(* CODESYS project mobject-graph-vision-pack.library
   Company: mobject
   Version: 0.5.0
   DefaultNamespace: mobject-graph-vision-pack
   Title: mobject-graph-vision-pack
   Placeholder: mobject-graph-vision-pack
   Author: mobject dev team
   DocFormat: reStructuredText

Project tree, tasks and I/O mapping:
  libraries: mobject-core, 0.3.0 (mobject); mobject-graph, 0.11.0 (mobject); mobject-graph-plc-pack, 0.12.0 (mobject); Tc2_Standard, * (Beckhoff Automation GmbH); Tc2_System, * (Beckhoff Automation GmbH); Tc3_Module, * (Beckhoff Automation GmbH); Tc3_Vision, * (Beckhoff Automation GmbH)
  Datatypes/
    Aliases/
    Arrays/
    Enums/
      function block _ETcVn2dCodeSearchStrategy [ST]: FB_init, AddLocalEnumeration, IsEnumeratorValueEqual, SetBaseDatatypeReference, Address, ClearReference, Clone, Identifier, MakeReferenceTo, Size, TryMakeReferenceTo, Value
      function block _ETcVnAdaptiveThresholdMethod [ST]: FB_init, AddLocalEnumeration, IsEnumeratorValueEqual, SetBaseDatatypeReference, Address, ClearReference, Clone, Identifier, MakeReferenceTo, Size, TryMakeReferenceTo, Value
      function block _ETcVnBarcodeSearchDirection [ST]: FB_init, AddLocalEnumeration, IsEnumeratorValueEqual, SetBaseDatatypeReference, Address, ClearReference, Clone, Identifier, MakeReferenceTo, Size, TryMakeReferenceTo, Value
      function block _ETcVnBarcodeType [ST]: FB_init, AddLocalEnumeration, IsEnumeratorValueEqual, SetBaseDatatypeReference, Address, ClearReference, Clone, Identifier, MakeReferenceTo, Size, TryMakeReferenceTo, Value
      function block _ETcVnBlobCombination [ST]: FB_init, AddLocalEnumeration, IsEnumeratorValueEqual, SetBaseDatatypeReference, Address, ClearReference, Clone, Identifier, MakeReferenceTo, Size, TryMakeReferenceTo, Value
      function block _ETcVnBorderInterpolationMethod [ST]: FB_init, AddLocalEnumeration, IsEnumeratorValueEqual, SetBaseDatatypeReference, Address, ClearReference, Clone, Identifier, MakeReferenceTo, Size, TryMakeReferenceTo, Value
      function block _ETcVnCalibrationPattern [ST]: FB_init, AddLocalEnumeration, IsEnumeratorValueEqual, SetBaseDatatypeReference, Address, ClearReference, Clone, Identifier, MakeReferenceTo, Size, TryMakeReferenceTo, Value
      function block _ETcVnCalibrationPatternOrigin [ST]: FB_init, AddLocalEnumeration, IsEnumeratorValueEqual, SetBaseDatatypeReference, Address, ClearReference, Clone, Identifier, MakeReferenceTo, Size, TryMakeReferenceTo, Value
      function block _ETcVnCameraState [ST]: FB_init, AddLocalEnumeration, IsEnumeratorValueEqual, SetBaseDatatypeReference, Address, ClearReference, Clone, Identifier, MakeReferenceTo, Size, TryMakeReferenceTo, Value
      function block _ETcVnClusteringAlgorithm [ST]: FB_init, AddLocalEnumeration, IsEnumeratorValueEqual, SetBaseDatatypeReference, Address, ClearReference, Clone, Identifier, MakeReferenceTo, Size, TryMakeReferenceTo, Value
      function block _ETcVnColorMap [ST]: FB_init, AddLocalEnumeration, IsEnumeratorValueEqual, SetBaseDatatypeReference, Address, ClearReference, Clone, Identifier, MakeReferenceTo, Size, TryMakeReferenceTo, Value
      function block _ETcVnColorMapSize [ST]: FB_init, AddLocalEnumeration, IsEnumeratorValueEqual, SetBaseDatatypeReference, Address, ClearReference, Clone, Identifier, MakeReferenceTo, Size, TryMakeReferenceTo, Value
      function block _ETcVnColorSpaceTransform [ST]: FB_init, AddLocalEnumeration, IsEnumeratorValueEqual, SetBaseDatatypeReference, Address, ClearReference, Clone, Identifier, MakeReferenceTo, Size, TryMakeReferenceTo, Value
      function block _ETcVnColorTrainingMethod [ST]: FB_init, AddLocalEnumeration, IsEnumeratorValueEqual, SetBaseDatatypeReference, Address, ClearReference, Clone, Identifier, MakeReferenceTo, Size, TryMakeReferenceTo, Value
      function block _ETcVnConnectedComponentsAlgorithm [ST]: FB_init, AddLocalEnumeration, IsEnumeratorValueEqual, SetBaseDatatypeReference, Address, ClearReference, Clone, Identifier, MakeReferenceTo, Size, TryMakeReferenceTo, Value
      function block _ETcVnContainerExportFormat [ST]: FB_init, AddLocalEnumeration, IsEnumeratorValueEqual, SetBaseDatatypeReference, Address, ClearReference, Clone, Identifier, MakeReferenceTo, Size, TryMakeReferenceTo, Value
      function block _ETcVnContourApproximationMethod [ST]: FB_init, AddLocalEnumeration, IsEnumeratorValueEqual, SetBaseDatatypeReference, Address, ClearReference, Clone, Identifier, MakeReferenceTo, Size, TryMakeReferenceTo, Value
      function block _ETcVnContourRetrievalMode [ST]: FB_init, AddLocalEnumeration, IsEnumeratorValueEqual, SetBaseDatatypeReference, Address, ClearReference, Clone, Identifier, MakeReferenceTo, Size, TryMakeReferenceTo, Value
      function block _ETcVnContoursMatchComparisonMethod [ST]: FB_init, AddLocalEnumeration, IsEnumeratorValueEqual, SetBaseDatatypeReference, Address, ClearReference, Clone, Identifier, MakeReferenceTo, Size, TryMakeReferenceTo, Value
      function block _ETcVnDiffusivityTypeKAZE [ST]: FB_init, AddLocalEnumeration, IsEnumeratorValueEqual, SetBaseDatatypeReference, Address, ClearReference, Clone, Identifier, MakeReferenceTo, Size, TryMakeReferenceTo, Value
      function block _ETcVnDistanceTransformationLabel [ST]: FB_init, AddLocalEnumeration, IsEnumeratorValueEqual, SetBaseDatatypeReference, Address, ClearReference, Clone, Identifier, MakeReferenceTo, Size, TryMakeReferenceTo, Value
      function block _ETcVnDistanceTransformationMask [ST]: FB_init, AddLocalEnumeration, IsEnumeratorValueEqual, SetBaseDatatypeReference, Address, ClearReference, Clone, Identifier, MakeReferenceTo, Size, TryMakeReferenceTo, Value
      function block _ETcVnDistanceType [ST]: FB_init, AddLocalEnumeration, IsEnumeratorValueEqual, SetBaseDatatypeReference, Address, ClearReference, Clone, Identifier, MakeReferenceTo, Size, TryMakeReferenceTo, Value
      function block _ETcVnDrawMatchesFlags [ST]: FB_init, AddLocalEnumeration, IsEnumeratorValueEqual, SetBaseDatatypeReference, Address, ClearReference, Clone, Identifier, MakeReferenceTo, Size, TryMakeReferenceTo, Value
      function block _ETcVnDrawShape [ST]: FB_init, AddLocalEnumeration, IsEnumeratorValueEqual, SetBaseDatatypeReference, Address, ClearReference, Clone, Identifier, MakeReferenceTo, Size, TryMakeReferenceTo, Value
      function block _ETcVnEdgeDetectionAlgorithm [ST]: FB_init, AddLocalEnumeration, IsEnumeratorValueEqual, SetBaseDatatypeReference, Address, ClearReference, Clone, Identifier, MakeReferenceTo, Size, TryMakeReferenceTo, Value
      function block _ETcVnEdgeDirection [ST]: FB_init, AddLocalEnumeration, IsEnumeratorValueEqual, SetBaseDatatypeReference, Address, ClearReference, Clone, Identifier, MakeReferenceTo, Size, TryMakeReferenceTo, Value
      function block _ETcVnElementType [ST]: FB_init, AddLocalEnumeration, IsEnumeratorValueEqual, SetBaseDatatypeReference, Address, ClearReference, Clone, Identifier, MakeReferenceTo, Size, TryMakeReferenceTo, Value
      function block _ETcVnEstimationAlgorithm [ST]: FB_init, AddLocalEnumeration, IsEnumeratorValueEqual, SetBaseDatatypeReference, Address, ClearReference, Clone, Identifier, MakeReferenceTo, Size, TryMakeReferenceTo, Value
      function block _ETcVnExtremePointDirection [ST]: FB_init, AddLocalEnumeration, IsEnumeratorValueEqual, SetBaseDatatypeReference, Address, ClearReference, Clone, Identifier, MakeReferenceTo, Size, TryMakeReferenceTo, Value
      function block _ETcVnFeatureDescriptorTypeAKAZE [ST]: FB_init, AddLocalEnumeration, IsEnumeratorValueEqual, SetBaseDatatypeReference, Address, ClearReference, Clone, Identifier, MakeReferenceTo, Size, TryMakeReferenceTo, Value
      function block _ETcVnFeatureScoreTypeORB [ST]: FB_init, AddLocalEnumeration, IsEnumeratorValueEqual, SetBaseDatatypeReference, Address, ClearReference, Clone, Identifier, MakeReferenceTo, Size, TryMakeReferenceTo, Value
      function block _ETcVnFilterDirection [ST]: FB_init, AddLocalEnumeration, IsEnumeratorValueEqual, SetBaseDatatypeReference, Address, ClearReference, Clone, Identifier, MakeReferenceTo, Size, TryMakeReferenceTo, Value
      function block _ETcVnFlipAxis [ST]: FB_init, AddLocalEnumeration, IsEnumeratorValueEqual, SetBaseDatatypeReference, Address, ClearReference, Clone, Identifier, MakeReferenceTo, Size, TryMakeReferenceTo, Value
      function block _ETcVnFontType [ST]: FB_init, AddLocalEnumeration, IsEnumeratorValueEqual, SetBaseDatatypeReference, Address, ClearReference, Clone, Identifier, MakeReferenceTo, Size, TryMakeReferenceTo, Value
      function block _ETcVnHoughMethod [ST]: FB_init, AddLocalEnumeration, IsEnumeratorValueEqual, SetBaseDatatypeReference, Address, ClearReference, Clone, Identifier, MakeReferenceTo, Size, TryMakeReferenceTo, Value
      function block _ETcVnInterpolationType [ST]: FB_init, AddLocalEnumeration, IsEnumeratorValueEqual, SetBaseDatatypeReference, Address, ClearReference, Clone, Identifier, MakeReferenceTo, Size, TryMakeReferenceTo, Value
      function block _ETcVnKeypointDetectionTypeAGAST [ST]: FB_init, AddLocalEnumeration, IsEnumeratorValueEqual, SetBaseDatatypeReference, Address, ClearReference, Clone, Identifier, MakeReferenceTo, Size, TryMakeReferenceTo, Value
      function block _ETcVnKeypointDetectionTypeFAST [ST]: FB_init, AddLocalEnumeration, IsEnumeratorValueEqual, SetBaseDatatypeReference, Address, ClearReference, Clone, Identifier, MakeReferenceTo, Size, TryMakeReferenceTo, Value
      function block _ETcVnLineType [ST]: FB_init, AddLocalEnumeration, IsEnumeratorValueEqual, SetBaseDatatypeReference, Address, ClearReference, Clone, Identifier, MakeReferenceTo, Size, TryMakeReferenceTo, Value
      function block _ETcVnMorphologicalOperator [ST]: FB_init, AddLocalEnumeration, IsEnumeratorValueEqual, SetBaseDatatypeReference, Address, ClearReference, Clone, Identifier, MakeReferenceTo, Size, TryMakeReferenceTo, Value
      function block _ETcVnNormalizationType [ST]: FB_init, AddLocalEnumeration, IsEnumeratorValueEqual, SetBaseDatatypeReference, Address, ClearReference, Clone, Identifier, MakeReferenceTo, Size, TryMakeReferenceTo, Value
      function block _ETcVnOrientationMethod [ST]: FB_init, AddLocalEnumeration, IsEnumeratorValueEqual, SetBaseDatatypeReference, Address, ClearReference, Clone, Identifier, MakeReferenceTo, Size, TryMakeReferenceTo, Value
      function block _ETcVnPixelConnectivity [ST]: FB_init, AddLocalEnumeration, IsEnumeratorValueEqual, SetBaseDatatypeReference, Address, ClearReference, Clone, Identifier, MakeReferenceTo, Size, TryMakeReferenceTo, Value
      function block _ETcVnPixelEncoding [ST]: FB_init, AddLocalEnumeration, IsEnumeratorValueEqual, SetBaseDatatypeReference, Address, ClearReference, Clone, Identifier, MakeReferenceTo, Size, TryMakeReferenceTo, Value
      function block _ETcVnPixelPackMode [ST]: FB_init, AddLocalEnumeration, IsEnumeratorValueEqual, SetBaseDatatypeReference, Address, ClearReference, Clone, Identifier, MakeReferenceTo, Size, TryMakeReferenceTo, Value
      function block _ETcVnRectangleIntersection [ST]: FB_init, AddLocalEnumeration, IsEnumeratorValueEqual, SetBaseDatatypeReference, Address, ClearReference, Clone, Identifier, MakeReferenceTo, Size, TryMakeReferenceTo, Value
      function block _ETcVnRotationAngle [ST]: FB_init, AddLocalEnumeration, IsEnumeratorValueEqual, SetBaseDatatypeReference, Address, ClearReference, Clone, Identifier, MakeReferenceTo, Size, TryMakeReferenceTo, Value
      function block _ETcVnSignedNormalization [ST]: FB_init, AddLocalEnumeration, IsEnumeratorValueEqual, SetBaseDatatypeReference, Address, ClearReference, Clone, Identifier, MakeReferenceTo, Size, TryMakeReferenceTo, Value
      function block _ETcVnStructuringElementShape [ST]: FB_init, AddLocalEnumeration, IsEnumeratorValueEqual, SetBaseDatatypeReference, Address, ClearReference, Clone, Identifier, MakeReferenceTo, Size, TryMakeReferenceTo, Value
      function block _ETcVnTemplateMatchMethod [ST]: FB_init, AddLocalEnumeration, IsEnumeratorValueEqual, SetBaseDatatypeReference, Address, ClearReference, Clone, Identifier, MakeReferenceTo, Size, TryMakeReferenceTo, Value
      function block _ETcVnThresholdType [ST]: FB_init, AddLocalEnumeration, IsEnumeratorValueEqual, SetBaseDatatypeReference, Address, ClearReference, Clone, Identifier, MakeReferenceTo, Size, TryMakeReferenceTo, Value
      function block _ETcVnVectorCompareMethod [ST]: FB_init, AddLocalEnumeration, IsEnumeratorValueEqual, SetBaseDatatypeReference, Address, ClearReference, Clone, Identifier, MakeReferenceTo, Size, TryMakeReferenceTo, Value
      function block _ETcVnWorldCoordinateSystem [ST]: FB_init, AddLocalEnumeration, IsEnumeratorValueEqual, SetBaseDatatypeReference, Address, ClearReference, Clone, Identifier, MakeReferenceTo, Size, TryMakeReferenceTo, Value
      function block _ETcWatchdogAccumulationType [ST]: FB_init, AddLocalEnumeration, IsEnumeratorValueEqual, SetBaseDatatypeReference, Address, ClearReference, Clone, Identifier, MakeReferenceTo, Size, TryMakeReferenceTo, Value
      function block _GEV_CAMERA_STATE [ST]: FB_init, AddLocalEnumeration, IsEnumeratorValueEqual, SetBaseDatatypeReference, Address, ClearReference, Clone, Identifier, MakeReferenceTo, Size, TryMakeReferenceTo, Value
    Interface/
      function block _ITcVnImage [ST]: TryGetElementTypeFromInfo, Address, ClearReference, Clone, Identifier, MakeReferenceTo, SerializeWith, Size, TryDeserializeFrom, TryMakeReferenceTo, Value
    Structs/
      function block _TcVnImageInfo [ST]: FB_init, SetMemberReference, Address, ClearReference, Clone, Identifier, MakeReferenceTo, nHeight, nImageSize, nWidth, nXPadding, nYPadding, Size, stPixelFormat, TryMakeReferenceTo, Value
      function block _TcVnPixelFormat [ST]: FB_init, SetMemberReference, Address, bFloat, bPlanar, bSigned, bSupported, ClearReference, Clone, ePixelEncoding, ePixelPackMode, Identifier, MakeReferenceTo, nChannels, nElementSize, nTotalSize, Size, TryMakeReferenceTo, Value
    function block VisionDatatypePack [ST]: RegisterWithDatatypes
  Nodes/
    Image Filtering/
      function block Node_F_VN_GaussianFilter [ST]: FB_init, Clone, OnExecute
    function block VisionNodePack [ST]: RegisterWithNodeFactory
  function block VisionPack [ST]: RegisterWithDatatypes, RegisterWithNodeFactory
*)

// Datatypes/Enums/_ETcVn2dCodeSearchStrategy
{attribute 'linkalways'} 
{attribute 'no_explicit_call' := 'This FB is a CLASS and must be accessed using methods or properties'}
{attribute 'enable_dynamic_creation'}
FUNCTION_BLOCK _ETcVn2dCodeSearchStrategy EXTENDS EnumDatatypeBase
VAR
	localData : ETcVn2dCodeSearchStrategy;
	activeData : REFERENCE TO ETcVn2dCodeSearchStrategy;
	enumBaseDatatype : _UDINT(localData);
END_VAR

METHOD FB_init : BOOL
VAR_INPUT
	bInitRetains : BOOL; // if TRUE, the retain variables are initialized (warm start / cold start)
	bInCopyCode : BOOL;  // if TRUE, the instance afterwards gets moved into the copy code (online change)
	InitialValue : ETcVn2dCodeSearchStrategy;
END_VAR
localData := InitialValue;
AddBaseDatatype(enumBaseDatatype);
ClearReference();

AddLocalEnumeration('TCVN_CSS_DEFAULT', ETcVn2dCodeSearchStrategy.TCVN_CSS_DEFAULT);
AddLocalEnumeration('TCVN_CSS_FIRST_FLIPPED', ETcVn2dCodeSearchStrategy.TCVN_CSS_FIRST_FLIPPED);
AddLocalEnumeration('TCVN_CSS_FIRST_INVERTED', ETcVn2dCodeSearchStrategy.TCVN_CSS_FIRST_INVERTED);
AddLocalEnumeration('TCVN_CSS_FIRST_NOT_FLIPPED', ETcVn2dCodeSearchStrategy.TCVN_CSS_FIRST_NOT_FLIPPED);
AddLocalEnumeration('TCVN_CSS_FIRST_NOT_INVERTED', ETcVn2dCodeSearchStrategy.TCVN_CSS_FIRST_NOT_INVERTED);
AddLocalEnumeration('TCVN_CSS_ONLY_FLIPPED', ETcVn2dCodeSearchStrategy.TCVN_CSS_ONLY_FLIPPED);
AddLocalEnumeration('TCVN_CSS_ONLY_INVERTED', ETcVn2dCodeSearchStrategy.TCVN_CSS_ONLY_INVERTED);
AddLocalEnumeration('TCVN_CSS_ONLY_NOT_FLIPPED', ETcVn2dCodeSearchStrategy.TCVN_CSS_ONLY_NOT_FLIPPED);
AddLocalEnumeration('TCVN_CSS_ONLY_NOT_INVERTED', ETcVn2dCodeSearchStrategy.TCVN_CSS_ONLY_NOT_INVERTED);
END_METHOD

METHOD PRIVATE AddLocalEnumeration
VAR_INPUT
	Enumeration : T_MAXSTRING;
	Value : ETcVn2dCodeSearchStrategy;
END_VAR
AddEnumeration(Enumeration, Value);
END_METHOD

METHOD IsEnumeratorValueEqual : BOOL
VAR_INPUT
	Enumerator : I_KeyValueForwardEnumerator;
END_VAR
VAR
	storedValue : ETcVn2dCodeSearchStrategy;
END_VAR
IF NOT Enumerator.TryGet(storedValue) THEN
	RETURN;
END_IF

IsEnumeratorValueEqual := storedValue = activeData;
END_METHOD

METHOD PROTECTED SetBaseDatatypeReference
VAR_INPUT
END_VAR
enumBaseDatatype.MakeReferenceTo(activeData);
END_METHOD

PROPERTY PUBLIC Address : PVOID
GET
Address := ADR(activeData);
END_GET
END_PROPERTY

METHOD PUBLIC ClearReference
VAR_INPUT
END_VAR
activeData REF= localData;
SetBaseDatatypeReference();
END_METHOD

METHOD PUBLIC Clone : I_Datatype
VAR
    pClone : POINTER TO _ETcVn2dCodeSearchStrategy;
END_VAR
pClone := __NEW(_ETcVn2dCodeSearchStrategy(InitialValue := Value));
Clone := pClone^;
END_METHOD

PROPERTY PUBLIC Identifier : T_MAXSTRING
GET
Identifier := 'ETcVn2dCodeSearchStrategy';
END_GET
END_PROPERTY

METHOD PUBLIC MakeReferenceTo
VAR_INPUT
	ReferenceTarget : REFERENCE TO ETcVn2dCodeSearchStrategy;
END_VAR
activeData REF= ReferenceTarget;
SetBaseDatatypeReference();
END_METHOD

PROPERTY PUBLIC Size : UDINT
GET
Size := SIZEOF(activeData);
END_GET
END_PROPERTY

METHOD TryMakeReferenceTo : BOOL
VAR_INPUT
	Target : I_Datatype;
END_VAR
VAR
	targetAsEnum : I_EnumDatatype;
	pTargetData : POINTER TO ETcVn2dCodeSearchStrategy;
END_VAR
IF NOT Target.TryResolveAsEnumDatatype(targetAsEnum) THEN
	RETURN;
END_IF

IF targetAsEnum.Identifier <> Identifier THEN
	RETURN;
END_IF

pTargetData := Target.Address;
activeData REF= pTargetData^;
SetBaseDatatypeReference();
TryMakeReferenceTo := TRUE;
END_METHOD

PROPERTY PUBLIC Value : ETcVn2dCodeSearchStrategy
GET
Value := activeData;
END_GET
SET
activeData := Value;
END_SET
END_PROPERTY

END_FUNCTION_BLOCK

// Datatypes/Enums/_ETcVnAdaptiveThresholdMethod
{attribute 'linkalways'} 
{attribute 'no_explicit_call' := 'This FB is a CLASS and must be accessed using methods or properties'}
{attribute 'enable_dynamic_creation'}
FUNCTION_BLOCK _ETcVnAdaptiveThresholdMethod EXTENDS EnumDatatypeBase
VAR
	localData : ETcVnAdaptiveThresholdMethod;
	activeData : REFERENCE TO ETcVnAdaptiveThresholdMethod;
	enumBaseDatatype : _DINT(localData);
END_VAR

METHOD FB_init : BOOL
VAR_INPUT
	bInitRetains : BOOL; // if TRUE, the retain variables are initialized (warm start / cold start)
	bInCopyCode : BOOL;  // if TRUE, the instance afterwards gets moved into the copy code (online change)
	InitialValue : ETcVnAdaptiveThresholdMethod;
END_VAR
localData := InitialValue;
AddBaseDatatype(enumBaseDatatype);
ClearReference();

AddLocalEnumeration('TCVN_ATM_MEAN', ETcVnAdaptiveThresholdMethod.TCVN_ATM_MEAN);
AddLocalEnumeration('TCVN_ATM_GAUSSIAN', ETcVnAdaptiveThresholdMethod.TCVN_ATM_GAUSSIAN);
END_METHOD

METHOD PRIVATE AddLocalEnumeration
VAR_INPUT
	Enumeration : T_MAXSTRING;
	Value : ETcVnAdaptiveThresholdMethod;
END_VAR
AddEnumeration(Enumeration, Value);
END_METHOD

METHOD IsEnumeratorValueEqual : BOOL
VAR_INPUT
	Enumerator : I_KeyValueForwardEnumerator;
END_VAR
VAR
	storedValue : ETcVnAdaptiveThresholdMethod;
END_VAR
IF NOT Enumerator.TryGet(storedValue) THEN
	RETURN;
END_IF

IsEnumeratorValueEqual := storedValue = activeData;
END_METHOD

METHOD PROTECTED SetBaseDatatypeReference
VAR_INPUT
END_VAR
enumBaseDatatype.MakeReferenceTo(activeData);
END_METHOD

PROPERTY PUBLIC Address : PVOID
GET
Address := ADR(activeData);
END_GET
END_PROPERTY

METHOD PUBLIC ClearReference
VAR_INPUT
END_VAR
activeData REF= localData;
SetBaseDatatypeReference();
END_METHOD

METHOD PUBLIC Clone : I_Datatype
VAR
    pClone : POINTER TO _ETcVnAdaptiveThresholdMethod;
END_VAR
pClone := __NEW(_ETcVnAdaptiveThresholdMethod(InitialValue := Value));
Clone := pClone^;
END_METHOD

PROPERTY PUBLIC Identifier : T_MAXSTRING
GET
Identifier := 'ETcVnAdaptiveThresholdMethod';
END_GET
END_PROPERTY

METHOD PUBLIC MakeReferenceTo
VAR_INPUT
	ReferenceTarget : REFERENCE TO ETcVnAdaptiveThresholdMethod;
END_VAR
activeData REF= ReferenceTarget;
SetBaseDatatypeReference();
END_METHOD

PROPERTY PUBLIC Size : UDINT
GET
Size := SIZEOF(activeData);
END_GET
END_PROPERTY

METHOD TryMakeReferenceTo : BOOL
VAR_INPUT
	Target : I_Datatype;
END_VAR
VAR
	targetAsEnum : I_EnumDatatype;
	pTargetData : POINTER TO ETcVnAdaptiveThresholdMethod;
END_VAR
IF NOT Target.TryResolveAsEnumDatatype(targetAsEnum) THEN
	RETURN;
END_IF

IF targetAsEnum.Identifier <> Identifier THEN
	RETURN;
END_IF

pTargetData := Target.Address;
activeData REF= pTargetData^;
SetBaseDatatypeReference();
TryMakeReferenceTo := TRUE;
END_METHOD

PROPERTY PUBLIC Value : ETcVnAdaptiveThresholdMethod
GET
Value := activeData;
END_GET
SET
activeData := Value;
END_SET
END_PROPERTY

END_FUNCTION_BLOCK

// Datatypes/Enums/_ETcVnBarcodeSearchDirection
{attribute 'linkalways'} 
{attribute 'no_explicit_call' := 'This FB is a CLASS and must be accessed using methods or properties'}
{attribute 'enable_dynamic_creation'}
FUNCTION_BLOCK _ETcVnBarcodeSearchDirection EXTENDS EnumDatatypeBase
VAR
	localData : ETcVnBarcodeSearchDirection;
	activeData : REFERENCE TO ETcVnBarcodeSearchDirection;
	enumBaseDatatype : _UDINT(localData);
END_VAR

METHOD FB_init : BOOL
VAR_INPUT
	bInitRetains : BOOL; // if TRUE, the retain variables are initialized (warm start / cold start)
	bInCopyCode : BOOL;  // if TRUE, the instance afterwards gets moved into the copy code (online change)
	InitialValue : ETcVnBarcodeSearchDirection;
END_VAR
localData := InitialValue;
AddBaseDatatype(enumBaseDatatype);
ClearReference();

AddLocalEnumeration('TCVN_BSD_ANY', ETcVnBarcodeSearchDirection.TCVN_BSD_ANY);
AddLocalEnumeration('TCVN_BSD_HORIZONTAL', ETcVnBarcodeSearchDirection.TCVN_BSD_HORIZONTAL);
AddLocalEnumeration('TCVN_BSD_VERTICAL', ETcVnBarcodeSearchDirection.TCVN_BSD_VERTICAL);
END_METHOD

METHOD PRIVATE AddLocalEnumeration
VAR_INPUT
	Enumeration : T_MAXSTRING;
	Value : ETcVnBarcodeSearchDirection;
END_VAR
AddEnumeration(Enumeration, Value);
END_METHOD

METHOD IsEnumeratorValueEqual : BOOL
VAR_INPUT
	Enumerator : I_KeyValueForwardEnumerator;
END_VAR
VAR
	storedValue : ETcVnBarcodeSearchDirection;
END_VAR
IF NOT Enumerator.TryGet(storedValue) THEN
	RETURN;
END_IF

IsEnumeratorValueEqual := storedValue = activeData;
END_METHOD

METHOD PROTECTED SetBaseDatatypeReference
VAR_INPUT
END_VAR
enumBaseDatatype.MakeReferenceTo(activeData);
END_METHOD

PROPERTY PUBLIC Address : PVOID
GET
Address := ADR(activeData);
END_GET
END_PROPERTY

METHOD PUBLIC ClearReference
VAR_INPUT
END_VAR
activeData REF= localData;
SetBaseDatatypeReference();
END_METHOD

METHOD PUBLIC Clone : I_Datatype
VAR
    pClone : POINTER TO _ETcVnBarcodeSearchDirection;
END_VAR
pClone := __NEW(_ETcVnBarcodeSearchDirection(InitialValue := Value));
Clone := pClone^;
END_METHOD

PROPERTY PUBLIC Identifier : T_MAXSTRING
GET
Identifier := 'ETcVnBarcodeSearchDirection';
END_GET
END_PROPERTY

METHOD PUBLIC MakeReferenceTo
VAR_INPUT
	ReferenceTarget : REFERENCE TO ETcVnBarcodeSearchDirection;
END_VAR
activeData REF= ReferenceTarget;
SetBaseDatatypeReference();
END_METHOD

PROPERTY PUBLIC Size : UDINT
GET
Size := SIZEOF(activeData);
END_GET
END_PROPERTY

METHOD TryMakeReferenceTo : BOOL
VAR_INPUT
	Target : I_Datatype;
END_VAR
VAR
	targetAsEnum : I_EnumDatatype;
	pTargetData : POINTER TO ETcVnBarcodeSearchDirection;
END_VAR
IF NOT Target.TryResolveAsEnumDatatype(targetAsEnum) THEN
	RETURN;
END_IF

IF targetAsEnum.Identifier <> Identifier THEN
	RETURN;
END_IF

pTargetData := Target.Address;
activeData REF= pTargetData^;
SetBaseDatatypeReference();
TryMakeReferenceTo := TRUE;
END_METHOD

PROPERTY PUBLIC Value : ETcVnBarcodeSearchDirection
GET
Value := activeData;
END_GET
SET
activeData := Value;
END_SET
END_PROPERTY

END_FUNCTION_BLOCK

// Datatypes/Enums/_ETcVnBarcodeType
{attribute 'linkalways'} 
{attribute 'no_explicit_call' := 'This FB is a CLASS and must be accessed using methods or properties'}
{attribute 'enable_dynamic_creation'}
FUNCTION_BLOCK _ETcVnBarcodeType EXTENDS EnumDatatypeBase
VAR
	localData : ETcVnBarcodeType;
	activeData : REFERENCE TO ETcVnBarcodeType;
	enumBaseDatatype : _UDINT(localData);
END_VAR

METHOD FB_init : BOOL
VAR_INPUT
	bInitRetains : BOOL; // if TRUE, the retain variables are initialized (warm start / cold start)
	bInCopyCode : BOOL;  // if TRUE, the instance afterwards gets moved into the copy code (online change)
	InitialValue : ETcVnBarcodeType;
END_VAR
localData := InitialValue;
AddBaseDatatype(enumBaseDatatype);
ClearReference();

AddLocalEnumeration('TCVN_BT_CODABAR', ETcVnBarcodeType.TCVN_BT_CODABAR);
AddLocalEnumeration('TCVN_BT_CODE39', ETcVnBarcodeType.TCVN_BT_CODE39);
AddLocalEnumeration('TCVN_BT_CODE93', ETcVnBarcodeType.TCVN_BT_CODE93);
AddLocalEnumeration('TCVN_BT_CODE128', ETcVnBarcodeType.TCVN_BT_CODE128);
AddLocalEnumeration('TCVN_BT_EAN8', ETcVnBarcodeType.TCVN_BT_EAN8);
AddLocalEnumeration('TCVN_BT_EAN13', ETcVnBarcodeType.TCVN_BT_EAN13);
AddLocalEnumeration('TCVN_BT_ITF', ETcVnBarcodeType.TCVN_BT_ITF);
AddLocalEnumeration('TCVN_BT_UPCA', ETcVnBarcodeType.TCVN_BT_UPCA);
AddLocalEnumeration('TCVN_BT_UPCE', ETcVnBarcodeType.TCVN_BT_UPCE);
AddLocalEnumeration('TCVN_BT_ANY', ETcVnBarcodeType.TCVN_BT_ANY);
AddLocalEnumeration('TCVN_BT_CODE39EXTENDED', ETcVnBarcodeType.TCVN_BT_CODE39EXTENDED);
END_METHOD

METHOD PRIVATE AddLocalEnumeration
VAR_INPUT
	Enumeration : T_MAXSTRING;
	Value : ETcVnBarcodeType;
END_VAR
AddEnumeration(Enumeration, Value);
END_METHOD

METHOD IsEnumeratorValueEqual : BOOL
VAR_INPUT
	Enumerator : I_KeyValueForwardEnumerator;
END_VAR
VAR
	storedValue : ETcVnBarcodeType;
END_VAR
IF NOT Enumerator.TryGet(storedValue) THEN
	RETURN;
END_IF

IsEnumeratorValueEqual := storedValue = activeData;
END_METHOD

METHOD PROTECTED SetBaseDatatypeReference
VAR_INPUT
END_VAR
enumBaseDatatype.MakeReferenceTo(activeData);
END_METHOD

PROPERTY PUBLIC Address : PVOID
GET
Address := ADR(activeData);
END_GET
END_PROPERTY

METHOD PUBLIC ClearReference
VAR_INPUT
END_VAR
activeData REF= localData;
SetBaseDatatypeReference();
END_METHOD

METHOD PUBLIC Clone : I_Datatype
VAR
    pClone : POINTER TO _ETcVnBarcodeType;
END_VAR
pClone := __NEW(_ETcVnBarcodeType(InitialValue := Value));
Clone := pClone^;
END_METHOD

PROPERTY PUBLIC Identifier : T_MAXSTRING
GET
Identifier := 'ETcVnBarcodeType';
END_GET
END_PROPERTY

METHOD PUBLIC MakeReferenceTo
VAR_INPUT
	ReferenceTarget : REFERENCE TO ETcVnBarcodeType;
END_VAR
activeData REF= ReferenceTarget;
SetBaseDatatypeReference();
END_METHOD

PROPERTY PUBLIC Size : UDINT
GET
Size := SIZEOF(activeData);
END_GET
END_PROPERTY

METHOD TryMakeReferenceTo : BOOL
VAR_INPUT
	Target : I_Datatype;
END_VAR
VAR
	targetAsEnum : I_EnumDatatype;
	pTargetData : POINTER TO ETcVnBarcodeType;
END_VAR
IF NOT Target.TryResolveAsEnumDatatype(targetAsEnum) THEN
	RETURN;
END_IF

IF targetAsEnum.Identifier <> Identifier THEN
	RETURN;
END_IF

pTargetData := Target.Address;
activeData REF= pTargetData^;
SetBaseDatatypeReference();
TryMakeReferenceTo := TRUE;
END_METHOD

PROPERTY PUBLIC Value : ETcVnBarcodeType
GET
Value := activeData;
END_GET
SET
activeData := Value;
END_SET
END_PROPERTY

END_FUNCTION_BLOCK

// Datatypes/Enums/_ETcVnBlobCombination
{attribute 'linkalways'} 
{attribute 'no_explicit_call' := 'This FB is a CLASS and must be accessed using methods or properties'}
{attribute 'enable_dynamic_creation'}
FUNCTION_BLOCK _ETcVnBlobCombination EXTENDS EnumDatatypeBase
VAR
	localData : ETcVnBlobCombination;
	activeData : REFERENCE TO ETcVnBlobCombination;
	enumBaseDatatype : _DINT(localData);
END_VAR

METHOD FB_init : BOOL
VAR_INPUT
	bInitRetains : BOOL; // if TRUE, the retain variables are initialized (warm start / cold start)
	bInCopyCode : BOOL;  // if TRUE, the instance afterwards gets moved into the copy code (online change)
	InitialValue : ETcVnBlobCombination;
END_VAR
localData := InitialValue;
AddBaseDatatype(enumBaseDatatype);
ClearReference();

AddLocalEnumeration('TCVN_BC_SMALLEST', ETcVnBlobCombination.TCVN_BC_SMALLEST);
AddLocalEnumeration('TCVN_BC_LARGEST', ETcVnBlobCombination.TCVN_BC_LARGEST);
AddLocalEnumeration('TCVN_BC_MIN_THRESHOLD', ETcVnBlobCombination.TCVN_BC_MIN_THRESHOLD);
AddLocalEnumeration('TCVN_BC_MAX_THRESHOLD', ETcVnBlobCombination.TCVN_BC_MAX_THRESHOLD);
AddLocalEnumeration('TCVN_BC_MEDIAN_THRESHOLD', ETcVnBlobCombination.TCVN_BC_MEDIAN_THRESHOLD);
END_METHOD

METHOD PRIVATE AddLocalEnumeration
VAR_INPUT
	Enumeration : T_MAXSTRING;
	Value : ETcVnBlobCombination;
END_VAR
AddEnumeration(Enumeration, Value);
END_METHOD

METHOD IsEnumeratorValueEqual : BOOL
VAR_INPUT
	Enumerator : I_KeyValueForwardEnumerator;
END_VAR
VAR
	storedValue : ETcVnBlobCombination;
END_VAR
IF NOT Enumerator.TryGet(storedValue) THEN
	RETURN;
END_IF

IsEnumeratorValueEqual := storedValue = activeData;
END_METHOD

METHOD PROTECTED SetBaseDatatypeReference
VAR_INPUT
END_VAR
enumBaseDatatype.MakeReferenceTo(activeData);
END_METHOD

PROPERTY PUBLIC Address : PVOID
GET
Address := ADR(activeData);
END_GET
END_PROPERTY

METHOD PUBLIC ClearReference
VAR_INPUT
END_VAR
activeData REF= localData;
SetBaseDatatypeReference();
END_METHOD

METHOD PUBLIC Clone : I_Datatype
VAR
    pClone : POINTER TO _ETcVnBlobCombination;
END_VAR
pClone := __NEW(_ETcVnBlobCombination(InitialValue := Value));
Clone := pClone^;
END_METHOD

PROPERTY PUBLIC Identifier : T_MAXSTRING
GET
Identifier := 'ETcVnBlobCombination';
END_GET
END_PROPERTY

METHOD PUBLIC MakeReferenceTo
VAR_INPUT
	ReferenceTarget : REFERENCE TO ETcVnBlobCombination;
END_VAR
activeData REF= ReferenceTarget;
SetBaseDatatypeReference();
END_METHOD

PROPERTY PUBLIC Size : UDINT
GET
Size := SIZEOF(activeData);
END_GET
END_PROPERTY

METHOD TryMakeReferenceTo : BOOL
VAR_INPUT
	Target : I_Datatype;
END_VAR
VAR
	targetAsEnum : I_EnumDatatype;
	pTargetData : POINTER TO ETcVnBlobCombination;
END_VAR
IF NOT Target.TryResolveAsEnumDatatype(targetAsEnum) THEN
	RETURN;
END_IF

IF targetAsEnum.Identifier <> Identifier THEN
	RETURN;
END_IF

pTargetData := Target.Address;
activeData REF= pTargetData^;
SetBaseDatatypeReference();
TryMakeReferenceTo := TRUE;
END_METHOD

PROPERTY PUBLIC Value : ETcVnBlobCombination
GET
Value := activeData;
END_GET
SET
activeData := Value;
END_SET
END_PROPERTY

END_FUNCTION_BLOCK

// Datatypes/Enums/_ETcVnBorderInterpolationMethod
{attribute 'linkalways'} 
{attribute 'no_explicit_call' := 'This FB is a CLASS and must be accessed using methods or properties'}
{attribute 'enable_dynamic_creation'}
FUNCTION_BLOCK _ETcVnBorderInterpolationMethod EXTENDS EnumDatatypeBase
VAR
	localData : ETcVnBorderInterpolationMethod;
	activeData : REFERENCE TO ETcVnBorderInterpolationMethod;
	enumBaseDatatype : _DINT(localData);
END_VAR

METHOD FB_init : BOOL
VAR_INPUT
	bInitRetains : BOOL; // if TRUE, the retain variables are initialized (warm start / cold start)
	bInCopyCode : BOOL;  // if TRUE, the instance afterwards gets moved into the copy code (online change)
	InitialValue : ETcVnBorderInterpolationMethod;
END_VAR
localData := InitialValue;
AddBaseDatatype(enumBaseDatatype);
ClearReference();

AddLocalEnumeration('TCVN_BIM_CONSTANT', ETcVnBorderInterpolationMethod.TCVN_BIM_CONSTANT);
AddLocalEnumeration('TCVN_BIM_REPLICATE', ETcVnBorderInterpolationMethod.TCVN_BIM_REPLICATE);
AddLocalEnumeration('TCVN_BIM_REFLECT', ETcVnBorderInterpolationMethod.TCVN_BIM_REFLECT);
AddLocalEnumeration('TCVN_BIM_WRAP', ETcVnBorderInterpolationMethod.TCVN_BIM_WRAP);
AddLocalEnumeration('TCVN_BIM_REFLECT_101', ETcVnBorderInterpolationMethod.TCVN_BIM_REFLECT_101);
AddLocalEnumeration('TCVN_BIM_DEFAULT', ETcVnBorderInterpolationMethod.TCVN_BIM_DEFAULT);
AddLocalEnumeration('TCVN_BIM_TRANSPARENT', ETcVnBorderInterpolationMethod.TCVN_BIM_TRANSPARENT);
AddLocalEnumeration('TCVN_BIM_ISOLATED_CONSTANT', ETcVnBorderInterpolationMethod.TCVN_BIM_ISOLATED_CONSTANT);
AddLocalEnumeration('TCVN_BIM_ISOLATED_REPLICATE', ETcVnBorderInterpolationMethod.TCVN_BIM_ISOLATED_REPLICATE);
AddLocalEnumeration('TCVN_BIM_ISOLATED_REFLECT', ETcVnBorderInterpolationMethod.TCVN_BIM_ISOLATED_REFLECT);
AddLocalEnumeration('TCVN_BIM_ISOLATED_WRAP', ETcVnBorderInterpolationMethod.TCVN_BIM_ISOLATED_WRAP);
AddLocalEnumeration('TCVN_BIM_ISOLATED_REFLECT_101', ETcVnBorderInterpolationMethod.TCVN_BIM_ISOLATED_REFLECT_101);
END_METHOD

METHOD PRIVATE AddLocalEnumeration
VAR_INPUT
	Enumeration : T_MAXSTRING;
	Value : ETcVnBorderInterpolationMethod;
END_VAR
AddEnumeration(Enumeration, Value);
END_METHOD

METHOD IsEnumeratorValueEqual : BOOL
VAR_INPUT
	Enumerator : I_KeyValueForwardEnumerator;
END_VAR
VAR
	storedValue : ETcVnBorderInterpolationMethod;
END_VAR
IF NOT Enumerator.TryGet(storedValue) THEN
	RETURN;
END_IF

IsEnumeratorValueEqual := storedValue = activeData;
END_METHOD

METHOD PROTECTED SetBaseDatatypeReference
VAR_INPUT
END_VAR
enumBaseDatatype.MakeReferenceTo(activeData);
END_METHOD

PROPERTY PUBLIC Address : PVOID
GET
Address := ADR(activeData);
END_GET
END_PROPERTY

METHOD PUBLIC ClearReference
VAR_INPUT
END_VAR
activeData REF= localData;
SetBaseDatatypeReference();
END_METHOD

METHOD PUBLIC Clone : I_Datatype
VAR
    pClone : POINTER TO _ETcVnBorderInterpolationMethod;
END_VAR
pClone := __NEW(_ETcVnBorderInterpolationMethod(InitialValue := Value));
Clone := pClone^;
END_METHOD

PROPERTY PUBLIC Identifier : T_MAXSTRING
GET
Identifier := 'ETcVnBorderInterpolationMethod';
END_GET
END_PROPERTY

METHOD PUBLIC MakeReferenceTo
VAR_INPUT
	ReferenceTarget : REFERENCE TO ETcVnBorderInterpolationMethod;
END_VAR
activeData REF= ReferenceTarget;
SetBaseDatatypeReference();
END_METHOD

PROPERTY PUBLIC Size : UDINT
GET
Size := SIZEOF(activeData);
END_GET
END_PROPERTY

METHOD TryMakeReferenceTo : BOOL
VAR_INPUT
	Target : I_Datatype;
END_VAR
VAR
	targetAsEnum : I_EnumDatatype;
	pTargetData : POINTER TO ETcVnBorderInterpolationMethod;
END_VAR
IF NOT Target.TryResolveAsEnumDatatype(targetAsEnum) THEN
	RETURN;
END_IF

IF targetAsEnum.Identifier <> Identifier THEN
	RETURN;
END_IF

pTargetData := Target.Address;
activeData REF= pTargetData^;
SetBaseDatatypeReference();
TryMakeReferenceTo := TRUE;
END_METHOD

PROPERTY PUBLIC Value : ETcVnBorderInterpolationMethod
GET
Value := activeData;
END_GET
SET
activeData := Value;
END_SET
END_PROPERTY

END_FUNCTION_BLOCK

// Datatypes/Enums/_ETcVnCalibrationPattern
{attribute 'linkalways'} 
{attribute 'no_explicit_call' := 'This FB is a CLASS and must be accessed using methods or properties'}
{attribute 'enable_dynamic_creation'}
FUNCTION_BLOCK _ETcVnCalibrationPattern EXTENDS EnumDatatypeBase
VAR
	localData : ETcVnCalibrationPattern;
	activeData : REFERENCE TO ETcVnCalibrationPattern;
	enumBaseDatatype : _DINT(localData);
END_VAR

METHOD FB_init : BOOL
VAR_INPUT
	bInitRetains : BOOL; // if TRUE, the retain variables are initialized (warm start / cold start)
	bInCopyCode : BOOL;  // if TRUE, the instance afterwards gets moved into the copy code (online change)
	InitialValue : ETcVnCalibrationPattern;
END_VAR
localData := InitialValue;
AddBaseDatatype(enumBaseDatatype);
ClearReference();

AddLocalEnumeration('TCVN_CP_CIRCLES_SYM', ETcVnCalibrationPattern.TCVN_CP_CIRCLES_SYM);
AddLocalEnumeration('TCVN_CP_CIRCLES_ASYM', ETcVnCalibrationPattern.TCVN_CP_CIRCLES_ASYM);
AddLocalEnumeration('TCVN_CP_CIRCLES_ASYM_INDENT', ETcVnCalibrationPattern.TCVN_CP_CIRCLES_ASYM_INDENT);
END_METHOD

METHOD PRIVATE AddLocalEnumeration
VAR_INPUT
	Enumeration : T_MAXSTRING;
	Value : ETcVnCalibrationPattern;
END_VAR
AddEnumeration(Enumeration, Value);
END_METHOD

METHOD IsEnumeratorValueEqual : BOOL
VAR_INPUT
	Enumerator : I_KeyValueForwardEnumerator;
END_VAR
VAR
	storedValue : ETcVnCalibrationPattern;
END_VAR
IF NOT Enumerator.TryGet(storedValue) THEN
	RETURN;
END_IF

IsEnumeratorValueEqual := storedValue = activeData;
END_METHOD

METHOD PROTECTED SetBaseDatatypeReference
VAR_INPUT
END_VAR
enumBaseDatatype.MakeReferenceTo(activeData);
END_METHOD

PROPERTY PUBLIC Address : PVOID
GET
Address := ADR(activeData);
END_GET
END_PROPERTY

METHOD PUBLIC ClearReference
VAR_INPUT
END_VAR
activeData REF= localData;
SetBaseDatatypeReference();
END_METHOD

METHOD PUBLIC Clone : I_Datatype
VAR
    pClone : POINTER TO _ETcVnCalibrationPattern;
END_VAR
pClone := __NEW(_ETcVnCalibrationPattern(InitialValue := Value));
Clone := pClone^;
END_METHOD

PROPERTY PUBLIC Identifier : T_MAXSTRING
GET
Identifier := 'ETcVnCalibrationPattern';
END_GET
END_PROPERTY

METHOD PUBLIC MakeReferenceTo
VAR_INPUT
	ReferenceTarget : REFERENCE TO ETcVnCalibrationPattern;
END_VAR
activeData REF= ReferenceTarget;
SetBaseDatatypeReference();
END_METHOD

PROPERTY PUBLIC Size : UDINT
GET
Size := SIZEOF(activeData);
END_GET
END_PROPERTY

METHOD TryMakeReferenceTo : BOOL
VAR_INPUT
	Target : I_Datatype;
END_VAR
VAR
	targetAsEnum : I_EnumDatatype;
	pTargetData : POINTER TO ETcVnCalibrationPattern;
END_VAR
IF NOT Target.TryResolveAsEnumDatatype(targetAsEnum) THEN
	RETURN;
END_IF

IF targetAsEnum.Identifier <> Identifier THEN
	RETURN;
END_IF

pTargetData := Target.Address;
activeData REF= pTargetData^;
SetBaseDatatypeReference();
TryMakeReferenceTo := TRUE;
END_METHOD

PROPERTY PUBLIC Value : ETcVnCalibrationPattern
GET
Value := activeData;
END_GET
SET
activeData := Value;
END_SET
END_PROPERTY

END_FUNCTION_BLOCK

// Datatypes/Enums/_ETcVnCalibrationPatternOrigin
{attribute 'linkalways'} 
{attribute 'no_explicit_call' := 'This FB is a CLASS and must be accessed using methods or properties'}
{attribute 'enable_dynamic_creation'}
FUNCTION_BLOCK _ETcVnCalibrationPatternOrigin EXTENDS EnumDatatypeBase
VAR
	localData : ETcVnCalibrationPatternOrigin;
	activeData : REFERENCE TO ETcVnCalibrationPatternOrigin;
	enumBaseDatatype : _DINT(localData);
END_VAR

METHOD FB_init : BOOL
VAR_INPUT
	bInitRetains : BOOL; // if TRUE, the retain variables are initialized (warm start / cold start)
	bInCopyCode : BOOL;  // if TRUE, the instance afterwards gets moved into the copy code (online change)
	InitialValue : ETcVnCalibrationPatternOrigin;
END_VAR
localData := InitialValue;
AddBaseDatatype(enumBaseDatatype);
ClearReference();

AddLocalEnumeration('TCVN_CPO_TOPLEFT', ETcVnCalibrationPatternOrigin.TCVN_CPO_TOPLEFT);
AddLocalEnumeration('TCVN_CPO_TOPCENTER', ETcVnCalibrationPatternOrigin.TCVN_CPO_TOPCENTER);
AddLocalEnumeration('TCVN_CPO_TOPRIGHT', ETcVnCalibrationPatternOrigin.TCVN_CPO_TOPRIGHT);
AddLocalEnumeration('TCVN_CPO_CENTERLEFT', ETcVnCalibrationPatternOrigin.TCVN_CPO_CENTERLEFT);
AddLocalEnumeration('TCVN_CPO_CENTER', ETcVnCalibrationPatternOrigin.TCVN_CPO_CENTER);
AddLocalEnumeration('TCVN_CPO_CENTERRIGHT', ETcVnCalibrationPatternOrigin.TCVN_CPO_CENTERRIGHT);
AddLocalEnumeration('TCVN_CPO_BOTTOMLEFT', ETcVnCalibrationPatternOrigin.TCVN_CPO_BOTTOMLEFT);
AddLocalEnumeration('TCVN_CPO_BOTTOMCENTER', ETcVnCalibrationPatternOrigin.TCVN_CPO_BOTTOMCENTER);
AddLocalEnumeration('TCVN_CPO_BOTTOMRIGHT', ETcVnCalibrationPatternOrigin.TCVN_CPO_BOTTOMRIGHT);
END_METHOD

METHOD PRIVATE AddLocalEnumeration
VAR_INPUT
	Enumeration : T_MAXSTRING;
	Value : ETcVnCalibrationPatternOrigin;
END_VAR
AddEnumeration(Enumeration, Value);
END_METHOD

METHOD IsEnumeratorValueEqual : BOOL
VAR_INPUT
	Enumerator : I_KeyValueForwardEnumerator;
END_VAR
VAR
	storedValue : ETcVnCalibrationPatternOrigin;
END_VAR
IF NOT Enumerator.TryGet(storedValue) THEN
	RETURN;
END_IF

IsEnumeratorValueEqual := storedValue = activeData;
END_METHOD

METHOD PROTECTED SetBaseDatatypeReference
VAR_INPUT
END_VAR
enumBaseDatatype.MakeReferenceTo(activeData);
END_METHOD

PROPERTY PUBLIC Address : PVOID
GET
Address := ADR(activeData);
END_GET
END_PROPERTY

METHOD PUBLIC ClearReference
VAR_INPUT
END_VAR
activeData REF= localData;
SetBaseDatatypeReference();
END_METHOD

METHOD PUBLIC Clone : I_Datatype
VAR
    pClone : POINTER TO _ETcVnCalibrationPatternOrigin;
END_VAR
pClone := __NEW(_ETcVnCalibrationPatternOrigin(InitialValue := Value));
Clone := pClone^;
END_METHOD

PROPERTY PUBLIC Identifier : T_MAXSTRING
GET
Identifier := 'ETcVnCalibrationPatternOrigin';
END_GET
END_PROPERTY

METHOD PUBLIC MakeReferenceTo
VAR_INPUT
	ReferenceTarget : REFERENCE TO ETcVnCalibrationPatternOrigin;
END_VAR
activeData REF= ReferenceTarget;
SetBaseDatatypeReference();
END_METHOD

PROPERTY PUBLIC Size : UDINT
GET
Size := SIZEOF(activeData);
END_GET
END_PROPERTY

METHOD TryMakeReferenceTo : BOOL
VAR_INPUT
	Target : I_Datatype;
END_VAR
VAR
	targetAsEnum : I_EnumDatatype;
	pTargetData : POINTER TO ETcVnCalibrationPatternOrigin;
END_VAR
IF NOT Target.TryResolveAsEnumDatatype(targetAsEnum) THEN
	RETURN;
END_IF

IF targetAsEnum.Identifier <> Identifier THEN
	RETURN;
END_IF

pTargetData := Target.Address;
activeData REF= pTargetData^;
SetBaseDatatypeReference();
TryMakeReferenceTo := TRUE;
END_METHOD

PROPERTY PUBLIC Value : ETcVnCalibrationPatternOrigin
GET
Value := activeData;
END_GET
SET
activeData := Value;
END_SET
END_PROPERTY

END_FUNCTION_BLOCK

// Datatypes/Enums/_ETcVnCameraState
{attribute 'linkalways'} 
{attribute 'no_explicit_call' := 'This FB is a CLASS and must be accessed using methods or properties'}
{attribute 'enable_dynamic_creation'}
FUNCTION_BLOCK _ETcVnCameraState EXTENDS EnumDatatypeBase
VAR
	localData : ETcVnCameraState;
	activeData : REFERENCE TO ETcVnCameraState;
	enumBaseDatatype : _DINT(localData);
END_VAR

METHOD FB_init : BOOL
VAR_INPUT
	bInitRetains : BOOL; // if TRUE, the retain variables are initialized (warm start / cold start)
	bInCopyCode : BOOL;  // if TRUE, the instance afterwards gets moved into the copy code (online change)
	InitialValue : ETcVnCameraState;
END_VAR
localData := InitialValue;
AddBaseDatatype(enumBaseDatatype);
ClearReference();

AddLocalEnumeration('TCVN_CS_ERROR', ETcVnCameraState.TCVN_CS_ERROR);
AddLocalEnumeration('TCVN_CS_INITIAL', ETcVnCameraState.TCVN_CS_INITIAL);
AddLocalEnumeration('TCVN_CS_INITIALIZING', ETcVnCameraState.TCVN_CS_INITIALIZING);
AddLocalEnumeration('TCVN_CS_INITIALIZED', ETcVnCameraState.TCVN_CS_INITIALIZED);
AddLocalEnumeration('TCVN_CS_OPENING', ETcVnCameraState.TCVN_CS_OPENING);
AddLocalEnumeration('TCVN_CS_OPENED', ETcVnCameraState.TCVN_CS_OPENED);
AddLocalEnumeration('TCVN_CS_STARTACQUISITION', ETcVnCameraState.TCVN_CS_STARTACQUISITION);
AddLocalEnumeration('TCVN_CS_ACQUIRING', ETcVnCameraState.TCVN_CS_ACQUIRING);
AddLocalEnumeration('TCVN_CS_STOPACQUISITION', ETcVnCameraState.TCVN_CS_STOPACQUISITION);
AddLocalEnumeration('TCVN_CS_RESETTINGFEATURES', ETcVnCameraState.TCVN_CS_RESETTINGFEATURES);
AddLocalEnumeration('TCVN_CS_TRIGGERING', ETcVnCameraState.TCVN_CS_TRIGGERING);
AddLocalEnumeration('TCVN_CS_CLOSING', ETcVnCameraState.TCVN_CS_CLOSING);
END_METHOD

METHOD PRIVATE AddLocalEnumeration
VAR_INPUT
	Enumeration : T_MAXSTRING;
	Value : ETcVnCameraState;
END_VAR
AddEnumeration(Enumeration, Value);
END_METHOD

METHOD IsEnumeratorValueEqual : BOOL
VAR_INPUT
	Enumerator : I_KeyValueForwardEnumerator;
END_VAR
VAR
	storedValue : ETcVnCameraState;
END_VAR
IF NOT Enumerator.TryGet(storedValue) THEN
	RETURN;
END_IF

IsEnumeratorValueEqual := storedValue = activeData;
END_METHOD

METHOD PROTECTED SetBaseDatatypeReference
VAR_INPUT
END_VAR
enumBaseDatatype.MakeReferenceTo(activeData);
END_METHOD

PROPERTY PUBLIC Address : PVOID
GET
Address := ADR(activeData);
END_GET
END_PROPERTY

METHOD PUBLIC ClearReference
VAR_INPUT
END_VAR
activeData REF= localData;
SetBaseDatatypeReference();
END_METHOD

METHOD PUBLIC Clone : I_Datatype
VAR
    pClone : POINTER TO _ETcVnCameraState;
END_VAR
pClone := __NEW(_ETcVnCameraState(InitialValue := Value));
Clone := pClone^;
END_METHOD

PROPERTY PUBLIC Identifier : T_MAXSTRING
GET
Identifier := 'ETcVnCameraState';
END_GET
END_PROPERTY

METHOD PUBLIC MakeReferenceTo
VAR_INPUT
	ReferenceTarget : REFERENCE TO ETcVnCalibrationPatternOrigin;
END_VAR
activeData REF= ReferenceTarget;
SetBaseDatatypeReference();
END_METHOD

PROPERTY PUBLIC Size : UDINT
GET
Size := SIZEOF(activeData);
END_GET
END_PROPERTY

METHOD TryMakeReferenceTo : BOOL
VAR_INPUT
	Target : I_Datatype;
END_VAR
VAR
	targetAsEnum : I_EnumDatatype;
	pTargetData : POINTER TO ETcVnCameraState;
END_VAR
IF NOT Target.TryResolveAsEnumDatatype(targetAsEnum) THEN
	RETURN;
END_IF

IF targetAsEnum.Identifier <> Identifier THEN
	RETURN;
END_IF

pTargetData := Target.Address;
activeData REF= pTargetData^;
SetBaseDatatypeReference();
TryMakeReferenceTo := TRUE;
END_METHOD

PROPERTY PUBLIC Value : ETcVnCameraState
GET
Value := activeData;
END_GET
SET
activeData := Value;
END_SET
END_PROPERTY

END_FUNCTION_BLOCK

// Datatypes/Enums/_ETcVnClusteringAlgorithm
{attribute 'linkalways'} 
{attribute 'no_explicit_call' := 'This FB is a CLASS and must be accessed using methods or properties'}
{attribute 'enable_dynamic_creation'}
FUNCTION_BLOCK _ETcVnClusteringAlgorithm EXTENDS EnumDatatypeBase
VAR
	localData : ETcVnClusteringAlgorithm;
	activeData : REFERENCE TO ETcVnClusteringAlgorithm;
	enumBaseDatatype : _DINT(localData);
END_VAR

METHOD FB_init : BOOL
VAR_INPUT
	bInitRetains : BOOL; // if TRUE, the retain variables are initialized (warm start / cold start)
	bInCopyCode : BOOL;  // if TRUE, the instance afterwards gets moved into the copy code (online change)
	InitialValue : ETcVnClusteringAlgorithm;
END_VAR
localData := InitialValue;
AddBaseDatatype(enumBaseDatatype);
ClearReference();

AddLocalEnumeration('TCVN_CA_KMEANSPP', ETcVnClusteringAlgorithm.TCVN_CA_KMEANSPP);
AddLocalEnumeration('TCVN_CA_LBG', ETcVnClusteringAlgorithm.TCVN_CA_LBG);
END_METHOD

METHOD PRIVATE AddLocalEnumeration
VAR_INPUT
	Enumeration : T_MAXSTRING;
	Value : ETcVnClusteringAlgorithm;
END_VAR
AddEnumeration(Enumeration, Value);
END_METHOD

METHOD IsEnumeratorValueEqual : BOOL
VAR_INPUT
	Enumerator : I_KeyValueForwardEnumerator;
END_VAR
VAR
	storedValue : ETcVnClusteringAlgorithm;
END_VAR
IF NOT Enumerator.TryGet(storedValue) THEN
	RETURN;
END_IF

IsEnumeratorValueEqual := storedValue = activeData;
END_METHOD

METHOD PROTECTED SetBaseDatatypeReference
VAR_INPUT
END_VAR
enumBaseDatatype.MakeReferenceTo(activeData);
END_METHOD

PROPERTY PUBLIC Address : PVOID
GET
Address := ADR(activeData);
END_GET
END_PROPERTY

METHOD PUBLIC ClearReference
VAR_INPUT
END_VAR
activeData REF= localData;
SetBaseDatatypeReference();
END_METHOD

METHOD PUBLIC Clone : I_Datatype
VAR
    pClone : POINTER TO _ETcVnClusteringAlgorithm;
END_VAR
pClone := __NEW(_ETcVnClusteringAlgorithm(InitialValue := Value));
Clone := pClone^;
END_METHOD

PROPERTY PUBLIC Identifier : T_MAXSTRING
GET
Identifier := 'ETcVnClusteringAlgorithm';
END_GET
END_PROPERTY

METHOD PUBLIC MakeReferenceTo
VAR_INPUT
	ReferenceTarget : REFERENCE TO ETcVnCalibrationPatternOrigin;
END_VAR
activeData REF= ReferenceTarget;
SetBaseDatatypeReference();
END_METHOD

PROPERTY PUBLIC Size : UDINT
GET
Size := SIZEOF(activeData);
END_GET
END_PROPERTY

METHOD TryMakeReferenceTo : BOOL
VAR_INPUT
	Target : I_Datatype;
END_VAR
VAR
	targetAsEnum : I_EnumDatatype;
	pTargetData : POINTER TO ETcVnClusteringAlgorithm;
END_VAR
IF NOT Target.TryResolveAsEnumDatatype(targetAsEnum) THEN
	RETURN;
END_IF

IF targetAsEnum.Identifier <> Identifier THEN
	RETURN;
END_IF

pTargetData := Target.Address;
activeData REF= pTargetData^;
SetBaseDatatypeReference();
TryMakeReferenceTo := TRUE;
END_METHOD

PROPERTY PUBLIC Value : ETcVnClusteringAlgorithm
GET
Value := activeData;
END_GET
SET
activeData := Value;
END_SET
END_PROPERTY

END_FUNCTION_BLOCK

// Datatypes/Enums/_ETcVnColorMap
{attribute 'linkalways'} 
{attribute 'no_explicit_call' := 'This FB is a CLASS and must be accessed using methods or properties'}
{attribute 'enable_dynamic_creation'}
FUNCTION_BLOCK _ETcVnColorMap EXTENDS EnumDatatypeBase
VAR
	localData : ETcVnColorMap;
	activeData : REFERENCE TO ETcVnColorMap;
	enumBaseDatatype : _DINT(localData);
END_VAR

METHOD FB_init : BOOL
VAR_INPUT
	bInitRetains : BOOL; // if TRUE, the retain variables are initialized (warm start / cold start)
	bInCopyCode : BOOL;  // if TRUE, the instance afterwards gets moved into the copy code (online change)
	InitialValue : ETcVnColorMap;
END_VAR
localData := InitialValue;
AddBaseDatatype(enumBaseDatatype);
ClearReference();

AddLocalEnumeration('TCVN_CM_AUTUMN', ETcVnColorMap.TCVN_CM_AUTUMN);
AddLocalEnumeration('TCVN_CM_BONE', ETcVnColorMap.TCVN_CM_BONE);
AddLocalEnumeration('TCVN_CM_JET', ETcVnColorMap.TCVN_CM_JET);
AddLocalEnumeration('TCVN_CM_WINTER', ETcVnColorMap.TCVN_CM_WINTER);
AddLocalEnumeration('TCVN_CM_RAINBOW', ETcVnColorMap.TCVN_CM_RAINBOW);
AddLocalEnumeration('TCVN_CM_OCEAN', ETcVnColorMap.TCVN_CM_OCEAN);
AddLocalEnumeration('TCVN_CM_SUMMER', ETcVnColorMap.TCVN_CM_SUMMER);
AddLocalEnumeration('TCVN_CM_SPRING', ETcVnColorMap.TCVN_CM_SPRING);
AddLocalEnumeration('TCVN_CM_COOL', ETcVnColorMap.TCVN_CM_COOL);
AddLocalEnumeration('TCVN_CM_HSV', ETcVnColorMap.TCVN_CM_HSV);
AddLocalEnumeration('TCVN_CM_PINK', ETcVnColorMap.TCVN_CM_PINK);
AddLocalEnumeration('TCVN_CM_HOT', ETcVnColorMap.TCVN_CM_HOT);
AddLocalEnumeration('TCVN_CM_PARULA', ETcVnColorMap.TCVN_CM_PARULA);
AddLocalEnumeration('TCVN_CM_MAGMA', ETcVnColorMap.TCVN_CM_MAGMA);
AddLocalEnumeration('TCVN_CM_INFERNO', ETcVnColorMap.TCVN_CM_INFERNO);
AddLocalEnumeration('TCVN_CM_PLASMA', ETcVnColorMap.TCVN_CM_PLASMA);
AddLocalEnumeration('TCVN_CM_VIRIDIS', ETcVnColorMap.TCVN_CM_VIRIDIS);
AddLocalEnumeration('TCVN_CM_CIVIDIS', ETcVnColorMap.TCVN_CM_CIVIDIS);
AddLocalEnumeration('TCVN_CM_TWILIGHT', ETcVnColorMap.TCVN_CM_TWILIGHT);
AddLocalEnumeration('TCVN_CM_TWILIGHT_SHIFTED', ETcVnColorMap.TCVN_CM_TWILIGHT_SHIFTED);
AddLocalEnumeration('TCVN_CM_TURBO', ETcVnColorMap.TCVN_CM_TURBO);
END_METHOD

METHOD PRIVATE AddLocalEnumeration
VAR_INPUT
	Enumeration : T_MAXSTRING;
	Value : ETcVnColorMap;
END_VAR
AddEnumeration(Enumeration, Value);
END_METHOD

METHOD IsEnumeratorValueEqual : BOOL
VAR_INPUT
	Enumerator : I_KeyValueForwardEnumerator;
END_VAR
VAR
	storedValue : ETcVnColorMap;
END_VAR
IF NOT Enumerator.TryGet(storedValue) THEN
	RETURN;
END_IF

IsEnumeratorValueEqual := storedValue = activeData;
END_METHOD

METHOD PROTECTED SetBaseDatatypeReference
VAR_INPUT
END_VAR
enumBaseDatatype.MakeReferenceTo(activeData);
END_METHOD

PROPERTY PUBLIC Address : PVOID
GET
Address := ADR(activeData);
END_GET
END_PROPERTY

METHOD PUBLIC ClearReference
VAR_INPUT
END_VAR
activeData REF= localData;
SetBaseDatatypeReference();
END_METHOD

METHOD PUBLIC Clone : I_Datatype
VAR
    pClone : POINTER TO _ETcVnColorMap;
END_VAR
pClone := __NEW(_ETcVnColorMap(InitialValue := Value));
Clone := pClone^;
END_METHOD

PROPERTY PUBLIC Identifier : T_MAXSTRING
GET
Identifier := 'ETcVnColorMap';
END_GET
END_PROPERTY

METHOD PUBLIC MakeReferenceTo
VAR_INPUT
	ReferenceTarget : REFERENCE TO ETcVnCalibrationPatternOrigin;
END_VAR
activeData REF= ReferenceTarget;
SetBaseDatatypeReference();
END_METHOD

PROPERTY PUBLIC Size : UDINT
GET
Size := SIZEOF(activeData);
END_GET
END_PROPERTY

METHOD TryMakeReferenceTo : BOOL
VAR_INPUT
	Target : I_Datatype;
END_VAR
VAR
	targetAsEnum : I_EnumDatatype;
	pTargetData : POINTER TO ETcVnColorMap;
END_VAR
IF NOT Target.TryResolveAsEnumDatatype(targetAsEnum) THEN
	RETURN;
END_IF

IF targetAsEnum.Identifier <> Identifier THEN
	RETURN;
END_IF

pTargetData := Target.Address;
activeData REF= pTargetData^;
SetBaseDatatypeReference();
TryMakeReferenceTo := TRUE;
END_METHOD

PROPERTY PUBLIC Value : ETcVnColorMap
GET
Value := activeData;
END_GET
SET
activeData := Value;
END_SET
END_PROPERTY

END_FUNCTION_BLOCK

// Datatypes/Enums/_ETcVnColorMapSize
{attribute 'linkalways'} 
{attribute 'no_explicit_call' := 'This FB is a CLASS and must be accessed using methods or properties'}
{attribute 'enable_dynamic_creation'}
FUNCTION_BLOCK _ETcVnColorMapSize EXTENDS EnumDatatypeBase
VAR
	localData : ETcVnColorMapSize;
	activeData : REFERENCE TO ETcVnColorMapSize;
	enumBaseDatatype : _UDINT(localData);
END_VAR

METHOD FB_init : BOOL
VAR_INPUT
	bInitRetains : BOOL; // if TRUE, the retain variables are initialized (warm start / cold start)
	bInCopyCode : BOOL;  // if TRUE, the instance afterwards gets moved into the copy code (online change)
	InitialValue : ETcVnColorMapSize;
END_VAR
localData := InitialValue;
AddBaseDatatype(enumBaseDatatype);
ClearReference();

AddLocalEnumeration('TCVN_CMS_256', ETcVnColorMapSize.TCVN_CMS_256);
AddLocalEnumeration('TCVN_CMS_65536', ETcVnColorMapSize.TCVN_CMS_65536);
END_METHOD

METHOD PRIVATE AddLocalEnumeration
VAR_INPUT
	Enumeration : T_MAXSTRING;
	Value : ETcVnColorMapSize;
END_VAR
AddEnumeration(Enumeration, Value);
END_METHOD

METHOD IsEnumeratorValueEqual : BOOL
VAR_INPUT
	Enumerator : I_KeyValueForwardEnumerator;
END_VAR
VAR
	storedValue : ETcVnColorMapSize;
END_VAR
IF NOT Enumerator.TryGet(storedValue) THEN
	RETURN;
END_IF

IsEnumeratorValueEqual := storedValue = activeData;
END_METHOD

METHOD PROTECTED SetBaseDatatypeReference
VAR_INPUT
END_VAR
enumBaseDatatype.MakeReferenceTo(activeData);
END_METHOD

PROPERTY PUBLIC Address : PVOID
GET
Address := ADR(activeData);
END_GET
END_PROPERTY

METHOD PUBLIC ClearReference
VAR_INPUT
END_VAR
activeData REF= localData;
SetBaseDatatypeReference();
END_METHOD

METHOD PUBLIC Clone : I_Datatype
VAR
    pClone : POINTER TO _ETcVnColorMapSize;
END_VAR
pClone := __NEW(_ETcVnColorMapSize(InitialValue := Value));
Clone := pClone^;
END_METHOD

PROPERTY PUBLIC Identifier : T_MAXSTRING
GET
Identifier := 'ETcVnColorMapSize';
END_GET
END_PROPERTY

METHOD PUBLIC MakeReferenceTo
VAR_INPUT
	ReferenceTarget : REFERENCE TO ETcVnColorMapSize;
END_VAR
activeData REF= ReferenceTarget;
SetBaseDatatypeReference();
END_METHOD

PROPERTY PUBLIC Size : UDINT
GET
Size := SIZEOF(activeData);
END_GET
END_PROPERTY

METHOD TryMakeReferenceTo : BOOL
VAR_INPUT
	Target : I_Datatype;
END_VAR
VAR
	targetAsEnum : I_EnumDatatype;
	pTargetData : POINTER TO ETcVnColorMapSize;
END_VAR
IF NOT Target.TryResolveAsEnumDatatype(targetAsEnum) THEN
	RETURN;
END_IF

IF targetAsEnum.Identifier <> Identifier THEN
	RETURN;
END_IF

pTargetData := Target.Address;
activeData REF= pTargetData^;
SetBaseDatatypeReference();
TryMakeReferenceTo := TRUE;
END_METHOD

PROPERTY PUBLIC Value : ETcVnColorMapSize
GET
Value := activeData;
END_GET
SET
activeData := Value;
END_SET
END_PROPERTY

END_FUNCTION_BLOCK

// Datatypes/Enums/_ETcVnColorSpaceTransform
{attribute 'linkalways'} 
{attribute 'no_explicit_call' := 'This FB is a CLASS and must be accessed using methods or properties'}
{attribute 'enable_dynamic_creation'}
FUNCTION_BLOCK _ETcVnColorSpaceTransform EXTENDS EnumDatatypeBase
VAR
	localData : ETcVnColorSpaceTransform;
	activeData : REFERENCE TO ETcVnColorSpaceTransform;
	enumBaseDatatype : _DINT(localData);
END_VAR

METHOD FB_init : BOOL
VAR_INPUT
	bInitRetains : BOOL; // if TRUE, the retain variables are initialized (warm start / cold start)
	bInCopyCode : BOOL;  // if TRUE, the instance afterwards gets moved into the copy code (online change)
	InitialValue : ETcVnColorSpaceTransform;
END_VAR
localData := InitialValue;
AddBaseDatatype(enumBaseDatatype);
ClearReference();

AddLocalEnumeration('TCVN_CST_BGR_TO_BGRA', ETcVnColorSpaceTransform.TCVN_CST_BGR_TO_BGRA);
AddLocalEnumeration('TCVN_CST_RGB_TO_RGBA', ETcVnColorSpaceTransform.TCVN_CST_RGB_TO_RGBA);
AddLocalEnumeration('TCVN_CST_BGRA_TO_BGR', ETcVnColorSpaceTransform.TCVN_CST_BGRA_TO_BGR);
AddLocalEnumeration('TCVN_CST_RGBA_TO_RGB', ETcVnColorSpaceTransform.TCVN_CST_RGBA_TO_RGB);
AddLocalEnumeration('TCVN_CST_BGR_TO_RGBA', ETcVnColorSpaceTransform.TCVN_CST_BGR_TO_RGBA);
AddLocalEnumeration('TCVN_CST_RGB_TO_BGRA', ETcVnColorSpaceTransform.TCVN_CST_RGB_TO_BGRA);
AddLocalEnumeration('TCVN_CST_BGRA_TO_RGB', ETcVnColorSpaceTransform.TCVN_CST_BGRA_TO_RGB);
AddLocalEnumeration('TCVN_CST_RGBA_TO_BGR', ETcVnColorSpaceTransform.TCVN_CST_RGBA_TO_BGR);
AddLocalEnumeration('TCVN_CST_BGR_TO_RGB', ETcVnColorSpaceTransform.TCVN_CST_BGR_TO_RGB);
AddLocalEnumeration('TCVN_CST_RGB_TO_BGR', ETcVnColorSpaceTransform.TCVN_CST_RGB_TO_BGR);
AddLocalEnumeration('TCVN_CST_BGRA_TO_RGBA', ETcVnColorSpaceTransform.TCVN_CST_BGRA_TO_RGBA);
AddLocalEnumeration('TCVN_CST_RGBA_TO_BGRA', ETcVnColorSpaceTransform.TCVN_CST_RGBA_TO_BGRA);
AddLocalEnumeration('TCVN_CST_BGR_TO_GRAY', ETcVnColorSpaceTransform.TCVN_CST_BGR_TO_GRAY);
AddLocalEnumeration('TCVN_CST_RGB_TO_GRAY', ETcVnColorSpaceTransform.TCVN_CST_RGB_TO_GRAY);
AddLocalEnumeration('TCVN_CST_GRAY_TO_BGR', ETcVnColorSpaceTransform.TCVN_CST_GRAY_TO_BGR);
AddLocalEnumeration('TCVN_CST_GRAY_TO_RGB', ETcVnColorSpaceTransform.TCVN_CST_GRAY_TO_RGB);
AddLocalEnumeration('TCVN_CST_GRAY_TO_BGRA', ETcVnColorSpaceTransform.TCVN_CST_GRAY_TO_BGRA);
AddLocalEnumeration('TCVN_CST_GRAY_TO_RGBA', ETcVnColorSpaceTransform.TCVN_CST_GRAY_TO_RGBA);
AddLocalEnumeration('TCVN_CST_BGRA_TO_GRAY', ETcVnColorSpaceTransform.TCVN_CST_BGRA_TO_GRAY);
AddLocalEnumeration('TCVN_CST_RGBA_TO_GRAY', ETcVnColorSpaceTransform.TCVN_CST_RGBA_TO_GRAY);
AddLocalEnumeration('TCVN_CST_RGB_TO_BGR_565', ETcVnColorSpaceTransform.TCVN_CST_RGB_TO_BGR_565);
AddLocalEnumeration('TCVN_CST_BGR_TO_BGR_565', ETcVnColorSpaceTransform.TCVN_CST_BGR_TO_BGR_565);
AddLocalEnumeration('TCVN_CST_BGR_565_TO_RGB', ETcVnColorSpaceTransform.TCVN_CST_BGR_565_TO_RGB);
AddLocalEnumeration('TCVN_CST_BGR_565_TO_BGR', ETcVnColorSpaceTransform.TCVN_CST_BGR_565_TO_BGR);
AddLocalEnumeration('TCVN_CST_RGBA_TO_BGR_565', ETcVnColorSpaceTransform.TCVN_CST_RGBA_TO_BGR_565);
AddLocalEnumeration('TCVN_CST_BGRA_TO_BGR_565', ETcVnColorSpaceTransform.TCVN_CST_BGRA_TO_BGR_565);
AddLocalEnumeration('TCVN_CST_BGR_565_TO_RGBA', ETcVnColorSpaceTransform.TCVN_CST_BGR_565_TO_RGBA);
AddLocalEnumeration('TCVN_CST_BGR_565_TO_BGRA', ETcVnColorSpaceTransform.TCVN_CST_BGR_565_TO_BGRA);
AddLocalEnumeration('TCVN_CST_GRAY_TO_BGR_565', ETcVnColorSpaceTransform.TCVN_CST_GRAY_TO_BGR_565);
AddLocalEnumeration('TCVN_CST_BGR_565_TO_GRAY', ETcVnColorSpaceTransform.TCVN_CST_BGR_565_TO_GRAY);
AddLocalEnumeration('TCVN_CST_RGB_TO_BGR_555', ETcVnColorSpaceTransform.TCVN_CST_RGB_TO_BGR_555);
AddLocalEnumeration('TCVN_CST_BGR_TO_BGR_555', ETcVnColorSpaceTransform.TCVN_CST_BGR_TO_BGR_555);
AddLocalEnumeration('TCVN_CST_BGR_555_TO_RGB', ETcVnColorSpaceTransform.TCVN_CST_BGR_555_TO_RGB);
AddLocalEnumeration('TCVN_CST_BGR_555_TO_BGR', ETcVnColorSpaceTransform.TCVN_CST_BGR_555_TO_BGR);
AddLocalEnumeration('TCVN_CST_RGBA_TO_BGR_555', ETcVnColorSpaceTransform.TCVN_CST_RGBA_TO_BGR_555);
AddLocalEnumeration('TCVN_CST_BGRA_TO_BGR_555', ETcVnColorSpaceTransform.TCVN_CST_BGRA_TO_BGR_555);
AddLocalEnumeration('TCVN_CST_BGR_555_TO_RGBA', ETcVnColorSpaceTransform.TCVN_CST_BGR_555_TO_RGBA);
AddLocalEnumeration('TCVN_CST_BGR_555_TO_BGRA', ETcVnColorSpaceTransform.TCVN_CST_BGR_555_TO_BGRA);
AddLocalEnumeration('TCVN_CST_GRAY_TO_BGR_555', ETcVnColorSpaceTransform.TCVN_CST_GRAY_TO_BGR_555);
AddLocalEnumeration('TCVN_CST_BGR_555_TO_GRAY', ETcVnColorSpaceTransform.TCVN_CST_BGR_555_TO_GRAY);
AddLocalEnumeration('TCVN_CST_BGR_TO_XYZ', ETcVnColorSpaceTransform.TCVN_CST_BGR_TO_XYZ);
AddLocalEnumeration('TCVN_CST_RGB_TO_XYZ', ETcVnColorSpaceTransform.TCVN_CST_RGB_TO_XYZ);
AddLocalEnumeration('TCVN_CST_XYZ_TO_BGR', ETcVnColorSpaceTransform.TCVN_CST_XYZ_TO_BGR);
AddLocalEnumeration('TCVN_CST_XYZ_TO_RGB', ETcVnColorSpaceTransform.TCVN_CST_XYZ_TO_RGB);
AddLocalEnumeration('TCVN_CST_BGR_TO_YCRCB', ETcVnColorSpaceTransform.TCVN_CST_BGR_TO_YCRCB);
AddLocalEnumeration('TCVN_CST_RGB_TO_YCRCB', ETcVnColorSpaceTransform.TCVN_CST_RGB_TO_YCRCB);
AddLocalEnumeration('TCVN_CST_YCRCB_TO_BGR', ETcVnColorSpaceTransform.TCVN_CST_YCRCB_TO_BGR);
AddLocalEnumeration('TCVN_CST_YCRCB_TO_RGB', ETcVnColorSpaceTransform.TCVN_CST_YCRCB_TO_RGB);
AddLocalEnumeration('TCVN_CST_BGR_TO_HSV', ETcVnColorSpaceTransform.TCVN_CST_BGR_TO_HSV);
AddLocalEnumeration('TCVN_CST_RGB_TO_HSV', ETcVnColorSpaceTransform.TCVN_CST_RGB_TO_HSV);
AddLocalEnumeration('TCVN_CST_BGR_TO_LAB', ETcVnColorSpaceTransform.TCVN_CST_BGR_TO_LAB);
AddLocalEnumeration('TCVN_CST_RGB_TO_LAB', ETcVnColorSpaceTransform.TCVN_CST_RGB_TO_LAB);
AddLocalEnumeration('TCVN_CST_BAYER_RG_TO_BGR', ETcVnColorSpaceTransform.TCVN_CST_BAYER_RG_TO_BGR);
AddLocalEnumeration('TCVN_CST_BAYER_BG_TO_RGB', ETcVnColorSpaceTransform.TCVN_CST_BAYER_BG_TO_RGB);
AddLocalEnumeration('TCVN_CST_BAYER_GR_TO_BGR', ETcVnColorSpaceTransform.TCVN_CST_BAYER_GR_TO_BGR);
AddLocalEnumeration('TCVN_CST_BAYER_GB_TO_RGB', ETcVnColorSpaceTransform.TCVN_CST_BAYER_GB_TO_RGB);
AddLocalEnumeration('TCVN_CST_BAYER_BG_TO_BGR', ETcVnColorSpaceTransform.TCVN_CST_BAYER_BG_TO_BGR);
AddLocalEnumeration('TCVN_CST_BAYER_RG_TO_RGB', ETcVnColorSpaceTransform.TCVN_CST_BAYER_RG_TO_RGB);
AddLocalEnumeration('TCVN_CST_BAYER_GB_TO_BGR', ETcVnColorSpaceTransform.TCVN_CST_BAYER_GB_TO_BGR);
AddLocalEnumeration('TCVN_CST_BAYER_GR_TO_RGB', ETcVnColorSpaceTransform.TCVN_CST_BAYER_GR_TO_RGB);
AddLocalEnumeration('TCVN_CST_BGR_TO_LUV', ETcVnColorSpaceTransform.TCVN_CST_BGR_TO_LUV);
AddLocalEnumeration('TCVN_CST_RGB_TO_LUV', ETcVnColorSpaceTransform.TCVN_CST_RGB_TO_LUV);
AddLocalEnumeration('TCVN_CST_BGR_TO_HLS', ETcVnColorSpaceTransform.TCVN_CST_BGR_TO_HLS);
AddLocalEnumeration('TCVN_CST_RGB_TO_HLS', ETcVnColorSpaceTransform.TCVN_CST_RGB_TO_HLS);
AddLocalEnumeration('TCVN_CST_HSV_TO_BGR', ETcVnColorSpaceTransform.TCVN_CST_HSV_TO_BGR);
AddLocalEnumeration('TCVN_CST_HSV_TO_RGB', ETcVnColorSpaceTransform.TCVN_CST_HSV_TO_RGB);
AddLocalEnumeration('TCVN_CST_LAB_TO_BGR', ETcVnColorSpaceTransform.TCVN_CST_LAB_TO_BGR);
AddLocalEnumeration('TCVN_CST_LAB_TO_RGB', ETcVnColorSpaceTransform.TCVN_CST_LAB_TO_RGB);
AddLocalEnumeration('TCVN_CST_LUV_TO_BGR', ETcVnColorSpaceTransform.TCVN_CST_LUV_TO_BGR);
AddLocalEnumeration('TCVN_CST_LUV_TO_RGB', ETcVnColorSpaceTransform.TCVN_CST_LUV_TO_RGB);
AddLocalEnumeration('TCVN_CST_HLS_TO_BGR', ETcVnColorSpaceTransform.TCVN_CST_HLS_TO_BGR);
AddLocalEnumeration('TCVN_CST_HLS_TO_RGB', ETcVnColorSpaceTransform.TCVN_CST_HLS_TO_RGB);
AddLocalEnumeration('TCVN_CST_BAYER_RG_TO_BGR_VNG', ETcVnColorSpaceTransform.TCVN_CST_BAYER_RG_TO_BGR_VNG);
AddLocalEnumeration('TCVN_CST_BAYER_GR_TO_BGR_VNG', ETcVnColorSpaceTransform.TCVN_CST_BAYER_GR_TO_BGR_VNG);
AddLocalEnumeration('TCVN_CST_BAYER_BG_TO_BGR_VNG', ETcVnColorSpaceTransform.TCVN_CST_BAYER_BG_TO_BGR_VNG);
AddLocalEnumeration('TCVN_CST_BAYER_GB_TO_BGR_VNG', ETcVnColorSpaceTransform.TCVN_CST_BAYER_GB_TO_BGR_VNG);
AddLocalEnumeration('TCVN_CST_BAYER_RG_TO_RGB_VNG', ETcVnColorSpaceTransform.TCVN_CST_BAYER_RG_TO_RGB_VNG);
AddLocalEnumeration('TCVN_CST_BAYER_GR_TO_RGB_VNG', ETcVnColorSpaceTransform.TCVN_CST_BAYER_GR_TO_RGB_VNG);
AddLocalEnumeration('TCVN_CST_BAYER_BG_TO_RGB_VNG', ETcVnColorSpaceTransform.TCVN_CST_BAYER_BG_TO_RGB_VNG);
AddLocalEnumeration('TCVN_CST_BAYER_GB_TO_RGB_VNG', ETcVnColorSpaceTransform.TCVN_CST_BAYER_GB_TO_RGB_VNG);
AddLocalEnumeration('TCVN_CST_BGR_TO_HSV_FULL', ETcVnColorSpaceTransform.TCVN_CST_BGR_TO_HSV_FULL);
AddLocalEnumeration('TCVN_CST_RGB_TO_HSV_FULL', ETcVnColorSpaceTransform.TCVN_CST_RGB_TO_HSV_FULL);
AddLocalEnumeration('TCVN_CST_BGR_TO_HLS_FULL', ETcVnColorSpaceTransform.TCVN_CST_BGR_TO_HLS_FULL);
AddLocalEnumeration('TCVN_CST_RGB_TO_HLS_FULL', ETcVnColorSpaceTransform.TCVN_CST_RGB_TO_HLS_FULL);
AddLocalEnumeration('TCVN_CST_HSV_TO_BGR_FULL', ETcVnColorSpaceTransform.TCVN_CST_HSV_TO_BGR_FULL);
AddLocalEnumeration('TCVN_CST_HSV_TO_RGB_FULL', ETcVnColorSpaceTransform.TCVN_CST_HSV_TO_RGB_FULL);
AddLocalEnumeration('TCVN_CST_HLS_TO_BGR_FULL', ETcVnColorSpaceTransform.TCVN_CST_HLS_TO_BGR_FULL);
AddLocalEnumeration('TCVN_CST_HLS_TO_RGB_FULL', ETcVnColorSpaceTransform.TCVN_CST_HLS_TO_RGB_FULL);
AddLocalEnumeration('TCVN_CST_LBGR_TO_LAB', ETcVnColorSpaceTransform.TCVN_CST_LBGR_TO_LAB);
AddLocalEnumeration('TCVN_CST_LRGB_TO_LAB', ETcVnColorSpaceTransform.TCVN_CST_LRGB_TO_LAB);
AddLocalEnumeration('TCVN_CST_LBGR_TO_LUV', ETcVnColorSpaceTransform.TCVN_CST_LBGR_TO_LUV);
AddLocalEnumeration('TCVN_CST_LRGB_TO_LUV', ETcVnColorSpaceTransform.TCVN_CST_LRGB_TO_LUV);
AddLocalEnumeration('TCVN_CST_LAB_TO_LBGR', ETcVnColorSpaceTransform.TCVN_CST_LAB_TO_LBGR);
AddLocalEnumeration('TCVN_CST_LAB_TO_LRGB', ETcVnColorSpaceTransform.TCVN_CST_LAB_TO_LRGB);
AddLocalEnumeration('TCVN_CST_LUV_TO_LBGR', ETcVnColorSpaceTransform.TCVN_CST_LUV_TO_LBGR);
AddLocalEnumeration('TCVN_CST_LUV_TO_LRGB', ETcVnColorSpaceTransform.TCVN_CST_LUV_TO_LRGB);
AddLocalEnumeration('TCVN_CST_BGR_TO_YUV', ETcVnColorSpaceTransform.TCVN_CST_BGR_TO_YUV);
AddLocalEnumeration('TCVN_CST_RGB_TO_YUV', ETcVnColorSpaceTransform.TCVN_CST_RGB_TO_YUV);
AddLocalEnumeration('TCVN_CST_YUV_TO_BGR', ETcVnColorSpaceTransform.TCVN_CST_YUV_TO_BGR);
AddLocalEnumeration('TCVN_CST_YUV_TO_RGB', ETcVnColorSpaceTransform.TCVN_CST_YUV_TO_RGB);
AddLocalEnumeration('TCVN_CST_BAYER_RG_TO_GRAY', ETcVnColorSpaceTransform.TCVN_CST_BAYER_RG_TO_GRAY);
AddLocalEnumeration('TCVN_CST_BAYER_GR_TO_GRAY', ETcVnColorSpaceTransform.TCVN_CST_BAYER_GR_TO_GRAY);
AddLocalEnumeration('TCVN_CST_BAYER_BG_TO_GRAY', ETcVnColorSpaceTransform.TCVN_CST_BAYER_BG_TO_GRAY);
AddLocalEnumeration('TCVN_CST_BAYER_GB_TO_GRAY', ETcVnColorSpaceTransform.TCVN_CST_BAYER_GB_TO_GRAY);
AddLocalEnumeration('TCVN_CST_YUV_420_NV12_TO_RGB', ETcVnColorSpaceTransform.TCVN_CST_YUV_420_NV12_TO_RGB);
AddLocalEnumeration('TCVN_CST_YUV_420_NV12_TO_BGR', ETcVnColorSpaceTransform.TCVN_CST_YUV_420_NV12_TO_BGR);
AddLocalEnumeration('TCVN_CST_YUV_420_NV21_TO_RGB', ETcVnColorSpaceTransform.TCVN_CST_YUV_420_NV21_TO_RGB);
AddLocalEnumeration('TCVN_CST_YUV_420_NV21_TO_BGR', ETcVnColorSpaceTransform.TCVN_CST_YUV_420_NV21_TO_BGR);
AddLocalEnumeration('TCVN_CST_YUV_420_SP_TO_RGB', ETcVnColorSpaceTransform.TCVN_CST_YUV_420_SP_TO_RGB);
AddLocalEnumeration('TCVN_CST_YUV_420_SP_TO_BGR', ETcVnColorSpaceTransform.TCVN_CST_YUV_420_SP_TO_BGR);
AddLocalEnumeration('TCVN_CST_YUV_420_NV12_TO_RGBA', ETcVnColorSpaceTransform.TCVN_CST_YUV_420_NV12_TO_RGBA);
AddLocalEnumeration('TCVN_CST_YUV_420_NV12_TO_BGRA', ETcVnColorSpaceTransform.TCVN_CST_YUV_420_NV12_TO_BGRA);
AddLocalEnumeration('TCVN_CST_YUV_420_NV21_TO_RGBA', ETcVnColorSpaceTransform.TCVN_CST_YUV_420_NV21_TO_RGBA);
AddLocalEnumeration('TCVN_CST_YUV_420_NV21_TO_BGRA', ETcVnColorSpaceTransform.TCVN_CST_YUV_420_NV21_TO_BGRA);
AddLocalEnumeration('TCVN_CST_YUV_420_SP_TO_RGBA', ETcVnColorSpaceTransform.TCVN_CST_YUV_420_SP_TO_RGBA);
AddLocalEnumeration('TCVN_CST_YUV_420_SP_TO_BGRA', ETcVnColorSpaceTransform.TCVN_CST_YUV_420_SP_TO_BGRA);
AddLocalEnumeration('TCVN_CST_YUV_420_YV12_TO_RGB', ETcVnColorSpaceTransform.TCVN_CST_YUV_420_YV12_TO_RGB);
AddLocalEnumeration('TCVN_CST_YUV_420_YV12_TO_BGR', ETcVnColorSpaceTransform.TCVN_CST_YUV_420_YV12_TO_BGR);
AddLocalEnumeration('TCVN_CST_YUV_420_IYUV_TO_RGB', ETcVnColorSpaceTransform.TCVN_CST_YUV_420_IYUV_TO_RGB);
AddLocalEnumeration('TCVN_CST_YUV_420_IYUV_TO_BGR', ETcVnColorSpaceTransform.TCVN_CST_YUV_420_IYUV_TO_BGR);
AddLocalEnumeration('TCVN_CST_YUV_420_I420_TO_RGB', ETcVnColorSpaceTransform.TCVN_CST_YUV_420_I420_TO_RGB);
AddLocalEnumeration('TCVN_CST_YUV_420_I420_TO_BGR', ETcVnColorSpaceTransform.TCVN_CST_YUV_420_I420_TO_BGR);
AddLocalEnumeration('TCVN_CST_YUV_420_P_TO_RGB', ETcVnColorSpaceTransform.TCVN_CST_YUV_420_P_TO_RGB);
AddLocalEnumeration('TCVN_CST_YUV_420_P_TO_BGR', ETcVnColorSpaceTransform.TCVN_CST_YUV_420_P_TO_BGR);
AddLocalEnumeration('TCVN_CST_YUV_420_YV12_TO_RGBA', ETcVnColorSpaceTransform.TCVN_CST_YUV_420_YV12_TO_RGBA);
AddLocalEnumeration('TCVN_CST_YUV_420_YV12_TO_BGRA', ETcVnColorSpaceTransform.TCVN_CST_YUV_420_YV12_TO_BGRA);
AddLocalEnumeration('TCVN_CST_YUV_420_IYUV_TO_RGBA', ETcVnColorSpaceTransform.TCVN_CST_YUV_420_IYUV_TO_RGBA);
AddLocalEnumeration('TCVN_CST_YUV_420_IYUV_TO_BGRA', ETcVnColorSpaceTransform.TCVN_CST_YUV_420_IYUV_TO_BGRA);
AddLocalEnumeration('TCVN_CST_YUV_420_I420_TO_RGBA', ETcVnColorSpaceTransform.TCVN_CST_YUV_420_I420_TO_RGBA);
AddLocalEnumeration('TCVN_CST_YUV_420_I420_TO_BGRA', ETcVnColorSpaceTransform.TCVN_CST_YUV_420_I420_TO_BGRA);
AddLocalEnumeration('TCVN_CST_YUV_420_P_TO_RGBA', ETcVnColorSpaceTransform.TCVN_CST_YUV_420_P_TO_RGBA);
AddLocalEnumeration('TCVN_CST_YUV_420_P_TO_BGRA', ETcVnColorSpaceTransform.TCVN_CST_YUV_420_P_TO_BGRA);
AddLocalEnumeration('TCVN_CST_YUV_420_TO_GRAY', ETcVnColorSpaceTransform.TCVN_CST_YUV_420_TO_GRAY);
AddLocalEnumeration('TCVN_CST_YUV_420_NV21_TO_GRAY', ETcVnColorSpaceTransform.TCVN_CST_YUV_420_NV21_TO_GRAY);
AddLocalEnumeration('TCVN_CST_YUV_420_NV12_TO_GRAY', ETcVnColorSpaceTransform.TCVN_CST_YUV_420_NV12_TO_GRAY);
AddLocalEnumeration('TCVN_CST_YUV_420_YV12_TO_GRAY', ETcVnColorSpaceTransform.TCVN_CST_YUV_420_YV12_TO_GRAY);
AddLocalEnumeration('TCVN_CST_YUV_420_IYUV_TO_GRAY', ETcVnColorSpaceTransform.TCVN_CST_YUV_420_IYUV_TO_GRAY);
AddLocalEnumeration('TCVN_CST_YUV_420_I420_TO_GRAY', ETcVnColorSpaceTransform.TCVN_CST_YUV_420_I420_TO_GRAY);
AddLocalEnumeration('TCVN_CST_YUV_420_SP_TO_GRAY', ETcVnColorSpaceTransform.TCVN_CST_YUV_420_SP_TO_GRAY);
AddLocalEnumeration('TCVN_CST_YUV_420_P_TO_GRAY', ETcVnColorSpaceTransform.TCVN_CST_YUV_420_P_TO_GRAY);
AddLocalEnumeration('TCVN_CST_YUV_422_UYVY_TO_RGB', ETcVnColorSpaceTransform.TCVN_CST_YUV_422_UYVY_TO_RGB);
AddLocalEnumeration('TCVN_CST_YUV_422_UYVY_TO_BGR', ETcVnColorSpaceTransform.TCVN_CST_YUV_422_UYVY_TO_BGR);
AddLocalEnumeration('TCVN_CST_YUV_422_Y422_TO_RGB', ETcVnColorSpaceTransform.TCVN_CST_YUV_422_Y422_TO_RGB);
AddLocalEnumeration('TCVN_CST_YUV_422_Y422_TO_BGR', ETcVnColorSpaceTransform.TCVN_CST_YUV_422_Y422_TO_BGR);
AddLocalEnumeration('TCVN_CST_YUV_422_UYNV_TO_RGB', ETcVnColorSpaceTransform.TCVN_CST_YUV_422_UYNV_TO_RGB);
AddLocalEnumeration('TCVN_CST_YUV_422_UYNV_TO_BGR', ETcVnColorSpaceTransform.TCVN_CST_YUV_422_UYNV_TO_BGR);
AddLocalEnumeration('TCVN_CST_YUV_422_UYVY_TO_RGBA', ETcVnColorSpaceTransform.TCVN_CST_YUV_422_UYVY_TO_RGBA);
AddLocalEnumeration('TCVN_CST_YUV_422_UYVY_TO_BGRA', ETcVnColorSpaceTransform.TCVN_CST_YUV_422_UYVY_TO_BGRA);
AddLocalEnumeration('TCVN_CST_YUV_422_Y422_TO_RGBA', ETcVnColorSpaceTransform.TCVN_CST_YUV_422_Y422_TO_RGBA);
AddLocalEnumeration('TCVN_CST_YUV_422_Y422_TO_BGRA', ETcVnColorSpaceTransform.TCVN_CST_YUV_422_Y422_TO_BGRA);
AddLocalEnumeration('TCVN_CST_YUV_422_UYNV_TO_RGBA', ETcVnColorSpaceTransform.TCVN_CST_YUV_422_UYNV_TO_RGBA);
AddLocalEnumeration('TCVN_CST_YUV_422_UYNV_TO_BGRA', ETcVnColorSpaceTransform.TCVN_CST_YUV_422_UYNV_TO_BGRA);
AddLocalEnumeration('TCVN_CST_YUV_422_YUY2_TO_RGB', ETcVnColorSpaceTransform.TCVN_CST_YUV_422_YUY2_TO_RGB);
AddLocalEnumeration('TCVN_CST_YUV_422_YUY2_TO_BGR', ETcVnColorSpaceTransform.TCVN_CST_YUV_422_YUY2_TO_BGR);
AddLocalEnumeration('TCVN_CST_YUV_422_YVYU_TO_RGB', ETcVnColorSpaceTransform.TCVN_CST_YUV_422_YVYU_TO_RGB);
AddLocalEnumeration('TCVN_CST_YUV_422_YVYU_TO_BGR', ETcVnColorSpaceTransform.TCVN_CST_YUV_422_YVYU_TO_BGR);
AddLocalEnumeration('TCVN_CST_YUV_422_YUYV_TO_RGB', ETcVnColorSpaceTransform.TCVN_CST_YUV_422_YUYV_TO_RGB);
AddLocalEnumeration('TCVN_CST_YUV_422_YUYV_TO_BGR', ETcVnColorSpaceTransform.TCVN_CST_YUV_422_YUYV_TO_BGR);
AddLocalEnumeration('TCVN_CST_YUV_422_YUNV_TO_RGB', ETcVnColorSpaceTransform.TCVN_CST_YUV_422_YUNV_TO_RGB);
AddLocalEnumeration('TCVN_CST_YUV_422_YUNV_TO_BGR', ETcVnColorSpaceTransform.TCVN_CST_YUV_422_YUNV_TO_BGR);
AddLocalEnumeration('TCVN_CST_YUV_422_YUY2_TO_RGBA', ETcVnColorSpaceTransform.TCVN_CST_YUV_422_YUY2_TO_RGBA);
AddLocalEnumeration('TCVN_CST_YUV_422_YUY2_TO_BGRA', ETcVnColorSpaceTransform.TCVN_CST_YUV_422_YUY2_TO_BGRA);
AddLocalEnumeration('TCVN_CST_YUV_422_YVYU_TO_RGBA', ETcVnColorSpaceTransform.TCVN_CST_YUV_422_YVYU_TO_RGBA);
AddLocalEnumeration('TCVN_CST_YUV_422_YVYU_TO_BGRA', ETcVnColorSpaceTransform.TCVN_CST_YUV_422_YVYU_TO_BGRA);
AddLocalEnumeration('TCVN_CST_YUV_422_YUYV_TO_RGBA', ETcVnColorSpaceTransform.TCVN_CST_YUV_422_YUYV_TO_RGBA);
AddLocalEnumeration('TCVN_CST_YUV_422_YUYV_TO_BGRA', ETcVnColorSpaceTransform.TCVN_CST_YUV_422_YUYV_TO_BGRA);
AddLocalEnumeration('TCVN_CST_YUV_422_YUNV_TO_RGBA', ETcVnColorSpaceTransform.TCVN_CST_YUV_422_YUNV_TO_RGBA);
AddLocalEnumeration('TCVN_CST_YUV_422_YUNV_TO_BGRA', ETcVnColorSpaceTransform.TCVN_CST_YUV_422_YUNV_TO_BGRA);
AddLocalEnumeration('TCVN_CST_YUV_422_UYVY_TO_GRAY', ETcVnColorSpaceTransform.TCVN_CST_YUV_422_UYVY_TO_GRAY);
AddLocalEnumeration('TCVN_CST_YUV_422_YUY2_TO_GRAY', ETcVnColorSpaceTransform.TCVN_CST_YUV_422_YUY2_TO_GRAY);
AddLocalEnumeration('TCVN_CST_YUV_422_Y422_TO_GRAY', ETcVnColorSpaceTransform.TCVN_CST_YUV_422_Y422_TO_GRAY);
AddLocalEnumeration('TCVN_CST_YUV_422_UYNV_TO_GRAY', ETcVnColorSpaceTransform.TCVN_CST_YUV_422_UYNV_TO_GRAY);
AddLocalEnumeration('TCVN_CST_YUV_422_YVYU_TO_GRAY', ETcVnColorSpaceTransform.TCVN_CST_YUV_422_YVYU_TO_GRAY);
AddLocalEnumeration('TCVN_CST_YUV_422_YUYV_TO_GRAY', ETcVnColorSpaceTransform.TCVN_CST_YUV_422_YUYV_TO_GRAY);
AddLocalEnumeration('TCVN_CST_YUV_422_YUNV_TO_GRAY', ETcVnColorSpaceTransform.TCVN_CST_YUV_422_YUNV_TO_GRAY);
AddLocalEnumeration('TCVN_CST_RGBA_TO_PREMULTIPLICATED_RGBA', ETcVnColorSpaceTransform.TCVN_CST_RGBA_TO_PREMULTIPLICATED_RGBA);
AddLocalEnumeration('TCVN_CST_PREMULTIPLICATED_RGBA_TO_RGBA', ETcVnColorSpaceTransform.TCVN_CST_PREMULTIPLICATED_RGBA_TO_RGBA);
AddLocalEnumeration('TCVN_CST_RGB_TO_YUV_420_I420', ETcVnColorSpaceTransform.TCVN_CST_RGB_TO_YUV_420_I420);
AddLocalEnumeration('TCVN_CST_BGR_TO_YUV_420_I420', ETcVnColorSpaceTransform.TCVN_CST_BGR_TO_YUV_420_I420);
AddLocalEnumeration('TCVN_CST_RGB_TO_YUV_420_IYUV', ETcVnColorSpaceTransform.TCVN_CST_RGB_TO_YUV_420_IYUV);
AddLocalEnumeration('TCVN_CST_BGR_TO_YUV_420_IYUV', ETcVnColorSpaceTransform.TCVN_CST_BGR_TO_YUV_420_IYUV);
AddLocalEnumeration('TCVN_CST_RGBA_TO_YUV_420_I420', ETcVnColorSpaceTransform.TCVN_CST_RGBA_TO_YUV_420_I420);
AddLocalEnumeration('TCVN_CST_BGRA_TO_YUV_420_I420', ETcVnColorSpaceTransform.TCVN_CST_BGRA_TO_YUV_420_I420);
AddLocalEnumeration('TCVN_CST_RGBA_TO_YUV_420_IYUV', ETcVnColorSpaceTransform.TCVN_CST_RGBA_TO_YUV_420_IYUV);
AddLocalEnumeration('TCVN_CST_BGRA_TO_YUV_420_IYUV', ETcVnColorSpaceTransform.TCVN_CST_BGRA_TO_YUV_420_IYUV);
AddLocalEnumeration('TCVN_CST_RGB_TO_YUV_420_YV12', ETcVnColorSpaceTransform.TCVN_CST_RGB_TO_YUV_420_YV12);
AddLocalEnumeration('TCVN_CST_BGR_TO_YUV_420_YV12', ETcVnColorSpaceTransform.TCVN_CST_BGR_TO_YUV_420_YV12);
AddLocalEnumeration('TCVN_CST_RGBA_TO_YUV_420_YV12', ETcVnColorSpaceTransform.TCVN_CST_RGBA_TO_YUV_420_YV12);
AddLocalEnumeration('TCVN_CST_BGRA_TO_YUV_420_YV12', ETcVnColorSpaceTransform.TCVN_CST_BGRA_TO_YUV_420_YV12);
AddLocalEnumeration('TCVN_CST_BAYER_RG_TO_BGR_EA', ETcVnColorSpaceTransform.TCVN_CST_BAYER_RG_TO_BGR_EA);
AddLocalEnumeration('TCVN_CST_BAYER_GR_TO_BGR_EA', ETcVnColorSpaceTransform.TCVN_CST_BAYER_GR_TO_BGR_EA);
AddLocalEnumeration('TCVN_CST_BAYER_BG_TO_BGR_EA', ETcVnColorSpaceTransform.TCVN_CST_BAYER_BG_TO_BGR_EA);
AddLocalEnumeration('TCVN_CST_BAYER_GB_TO_BGR_EA', ETcVnColorSpaceTransform.TCVN_CST_BAYER_GB_TO_BGR_EA);
AddLocalEnumeration('TCVN_CST_BAYER_RG_TO_RGB_EA', ETcVnColorSpaceTransform.TCVN_CST_BAYER_RG_TO_RGB_EA);
AddLocalEnumeration('TCVN_CST_BAYER_GR_TO_RGB_EA', ETcVnColorSpaceTransform.TCVN_CST_BAYER_GR_TO_RGB_EA);
AddLocalEnumeration('TCVN_CST_BAYER_BG_TO_RGB_EA', ETcVnColorSpaceTransform.TCVN_CST_BAYER_BG_TO_RGB_EA);
AddLocalEnumeration('TCVN_CST_BAYER_GB_TO_RGB_EA', ETcVnColorSpaceTransform.TCVN_CST_BAYER_GB_TO_RGB_EA);
AddLocalEnumeration('TCVN_CST_BAYER_RG_TO_BGRA', ETcVnColorSpaceTransform.TCVN_CST_BAYER_RG_TO_BGRA);
AddLocalEnumeration('TCVN_CST_BAYER_GR_TO_BGRA', ETcVnColorSpaceTransform.TCVN_CST_BAYER_GR_TO_BGRA);
AddLocalEnumeration('TCVN_CST_BAYER_BG_TO_BGRA', ETcVnColorSpaceTransform.TCVN_CST_BAYER_BG_TO_BGRA);
AddLocalEnumeration('TCVN_CST_BAYER_GB_TO_BGRA', ETcVnColorSpaceTransform.TCVN_CST_BAYER_GB_TO_BGRA);
AddLocalEnumeration('TCVN_CST_BAYER_RG_TO_RGBA', ETcVnColorSpaceTransform.TCVN_CST_BAYER_RG_TO_RGBA);
AddLocalEnumeration('TCVN_CST_BAYER_GR_TO_RGBA', ETcVnColorSpaceTransform.TCVN_CST_BAYER_GR_TO_RGBA);
AddLocalEnumeration('TCVN_CST_BAYER_BG_TO_RGBA', ETcVnColorSpaceTransform.TCVN_CST_BAYER_BG_TO_RGBA);
AddLocalEnumeration('TCVN_CST_BAYER_GB_TO_RGBA', ETcVnColorSpaceTransform.TCVN_CST_BAYER_GB_TO_RGBA);
AddLocalEnumeration('TCVN_CST_MAX', ETcVnColorSpaceTransform.TCVN_CST_MAX);
END_METHOD

METHOD PRIVATE AddLocalEnumeration
VAR_INPUT
	Enumeration : T_MAXSTRING;
	Value : ETcVnColorSpaceTransform;
END_VAR
AddEnumeration(Enumeration, Value);
END_METHOD

METHOD IsEnumeratorValueEqual : BOOL
VAR_INPUT
	Enumerator : I_KeyValueForwardEnumerator;
END_VAR
VAR
	storedValue : ETcVnColorSpaceTransform;
END_VAR
IF NOT Enumerator.TryGet(storedValue) THEN
	RETURN;
END_IF

IsEnumeratorValueEqual := storedValue = activeData;
END_METHOD

METHOD PROTECTED SetBaseDatatypeReference
VAR_INPUT
END_VAR
enumBaseDatatype.MakeReferenceTo(activeData);
END_METHOD

PROPERTY PUBLIC Address : PVOID
GET
Address := ADR(activeData);
END_GET
END_PROPERTY

METHOD PUBLIC ClearReference
VAR_INPUT
END_VAR
activeData REF= localData;
SetBaseDatatypeReference();
END_METHOD

METHOD PUBLIC Clone : I_Datatype
VAR
    pClone : POINTER TO _ETcVnColorSpaceTransform;
END_VAR
pClone := __NEW(_ETcVnColorSpaceTransform(InitialValue := Value));
Clone := pClone^;
END_METHOD

PROPERTY PUBLIC Identifier : T_MAXSTRING
GET
Identifier := 'ETcVnColorSpaceTransform';
END_GET
END_PROPERTY

METHOD PUBLIC MakeReferenceTo
VAR_INPUT
	ReferenceTarget : REFERENCE TO ETcVnColorSpaceTransform;
END_VAR
activeData REF= ReferenceTarget;
SetBaseDatatypeReference();
END_METHOD

PROPERTY PUBLIC Size : UDINT
GET
Size := SIZEOF(activeData);
END_GET
END_PROPERTY

METHOD TryMakeReferenceTo : BOOL
VAR_INPUT
	Target : I_Datatype;
END_VAR
VAR
	targetAsEnum : I_EnumDatatype;
	pTargetData : POINTER TO ETcVnColorSpaceTransform;
END_VAR
IF NOT Target.TryResolveAsEnumDatatype(targetAsEnum) THEN
	RETURN;
END_IF

IF targetAsEnum.Identifier <> Identifier THEN
	RETURN;
END_IF

pTargetData := Target.Address;
activeData REF= pTargetData^;
SetBaseDatatypeReference();
TryMakeReferenceTo := TRUE;
END_METHOD

PROPERTY PUBLIC Value : ETcVnColorSpaceTransform
GET
Value := activeData;
END_GET
SET
activeData := Value;
END_SET
END_PROPERTY

END_FUNCTION_BLOCK

// Datatypes/Enums/_ETcVnColorTrainingMethod
{attribute 'linkalways'} 
{attribute 'no_explicit_call' := 'This FB is a CLASS and must be accessed using methods or properties'}
{attribute 'enable_dynamic_creation'}
FUNCTION_BLOCK _ETcVnColorTrainingMethod EXTENDS EnumDatatypeBase
VAR
	localData : ETcVnColorTrainingMethod;
	activeData : REFERENCE TO ETcVnColorTrainingMethod;
	enumBaseDatatype : _DINT(localData);
END_VAR

METHOD FB_init : BOOL
VAR_INPUT
	bInitRetains : BOOL; // if TRUE, the retain variables are initialized (warm start / cold start)
	bInCopyCode : BOOL;  // if TRUE, the instance afterwards gets moved into the copy code (online change)
	InitialValue : ETcVnColorTrainingMethod;
END_VAR
localData := InitialValue;
AddBaseDatatype(enumBaseDatatype);
ClearReference();

AddLocalEnumeration('TCVN_CTM_LAB', ETcVnColorTrainingMethod.TCVN_CTM_LAB);
AddLocalEnumeration('TCVN_CTM_RGB', ETcVnColorTrainingMethod.TCVN_CTM_RGB);
END_METHOD

METHOD PRIVATE AddLocalEnumeration
VAR_INPUT
	Enumeration : T_MAXSTRING;
	Value : ETcVnColorTrainingMethod;
END_VAR
AddEnumeration(Enumeration, Value);
END_METHOD

METHOD IsEnumeratorValueEqual : BOOL
VAR_INPUT
	Enumerator : I_KeyValueForwardEnumerator;
END_VAR
VAR
	storedValue : ETcVnColorTrainingMethod;
END_VAR
IF NOT Enumerator.TryGet(storedValue) THEN
	RETURN;
END_IF

IsEnumeratorValueEqual := storedValue = activeData;
END_METHOD

METHOD PROTECTED SetBaseDatatypeReference
VAR_INPUT
END_VAR
enumBaseDatatype.MakeReferenceTo(activeData);
END_METHOD

PROPERTY PUBLIC Address : PVOID
GET
Address := ADR(activeData);
END_GET
END_PROPERTY

METHOD PUBLIC ClearReference
VAR_INPUT
END_VAR
activeData REF= localData;
SetBaseDatatypeReference();
END_METHOD

METHOD PUBLIC Clone : I_Datatype
VAR
    pClone : POINTER TO _ETcVnColorTrainingMethod;
END_VAR
pClone := __NEW(_ETcVnColorTrainingMethod(InitialValue := Value));
Clone := pClone^;
END_METHOD

PROPERTY PUBLIC Identifier : T_MAXSTRING
GET
Identifier := 'ETcVnColorTrainingMethod';
END_GET
END_PROPERTY

METHOD PUBLIC MakeReferenceTo
VAR_INPUT
	ReferenceTarget : REFERENCE TO ETcVnColorTrainingMethod;
END_VAR
activeData REF= ReferenceTarget;
SetBaseDatatypeReference();
END_METHOD

PROPERTY PUBLIC Size : UDINT
GET
Size := SIZEOF(activeData);
END_GET
END_PROPERTY

METHOD TryMakeReferenceTo : BOOL
VAR_INPUT
	Target : I_Datatype;
END_VAR
VAR
	targetAsEnum : I_EnumDatatype;
	pTargetData : POINTER TO ETcVnColorTrainingMethod;
END_VAR
IF NOT Target.TryResolveAsEnumDatatype(targetAsEnum) THEN
	RETURN;
END_IF

IF targetAsEnum.Identifier <> Identifier THEN
	RETURN;
END_IF

pTargetData := Target.Address;
activeData REF= pTargetData^;
SetBaseDatatypeReference();
TryMakeReferenceTo := TRUE;
END_METHOD

PROPERTY PUBLIC Value : ETcVnColorTrainingMethod
GET
Value := activeData;
END_GET
SET
activeData := Value;
END_SET
END_PROPERTY

END_FUNCTION_BLOCK

// Datatypes/Enums/_ETcVnConnectedComponentsAlgorithm
{attribute 'linkalways'} 
{attribute 'no_explicit_call' := 'This FB is a CLASS and must be accessed using methods or properties'}
{attribute 'enable_dynamic_creation'}
FUNCTION_BLOCK _ETcVnConnectedComponentsAlgorithm EXTENDS EnumDatatypeBase
VAR
	localData : ETcVnConnectedComponentsAlgorithm;
	activeData : REFERENCE TO ETcVnConnectedComponentsAlgorithm;
	enumBaseDatatype : _DINT(localData);
END_VAR

METHOD FB_init : BOOL
VAR_INPUT
	bInitRetains : BOOL; // if TRUE, the retain variables are initialized (warm start / cold start)
	bInCopyCode : BOOL;  // if TRUE, the instance afterwards gets moved into the copy code (online change)
	InitialValue : ETcVnConnectedComponentsAlgorithm;
END_VAR
localData := InitialValue;
AddBaseDatatype(enumBaseDatatype);
ClearReference();

AddLocalEnumeration('TCVN_CCA_WU', ETcVnConnectedComponentsAlgorithm.TCVN_CCA_WU);
AddLocalEnumeration('TCVN_CCA_GRANA', ETcVnConnectedComponentsAlgorithm.TCVN_CCA_GRANA);
END_METHOD

METHOD PRIVATE AddLocalEnumeration
VAR_INPUT
	Enumeration : T_MAXSTRING;
	Value : ETcVnConnectedComponentsAlgorithm;
END_VAR
AddEnumeration(Enumeration, Value);
END_METHOD

METHOD IsEnumeratorValueEqual : BOOL
VAR_INPUT
	Enumerator : I_KeyValueForwardEnumerator;
END_VAR
VAR
	storedValue : ETcVnConnectedComponentsAlgorithm;
END_VAR
IF NOT Enumerator.TryGet(storedValue) THEN
	RETURN;
END_IF

IsEnumeratorValueEqual := storedValue = activeData;
END_METHOD

METHOD PROTECTED SetBaseDatatypeReference
VAR_INPUT
END_VAR
enumBaseDatatype.MakeReferenceTo(activeData);
END_METHOD

PROPERTY PUBLIC Address : PVOID
GET
Address := ADR(activeData);
END_GET
END_PROPERTY

METHOD PUBLIC ClearReference
VAR_INPUT
END_VAR
activeData REF= localData;
SetBaseDatatypeReference();
END_METHOD

METHOD PUBLIC Clone : I_Datatype
VAR
    pClone : POINTER TO _ETcVnConnectedComponentsAlgorithm;
END_VAR
pClone := __NEW(_ETcVnConnectedComponentsAlgorithm(InitialValue := Value));
Clone := pClone^;
END_METHOD

PROPERTY PUBLIC Identifier : T_MAXSTRING
GET
Identifier := 'ETcVnConnectedComponentsAlgorithm';
END_GET
END_PROPERTY

METHOD PUBLIC MakeReferenceTo
VAR_INPUT
	ReferenceTarget : REFERENCE TO ETcVnConnectedComponentsAlgorithm;
END_VAR
activeData REF= ReferenceTarget;
SetBaseDatatypeReference();
END_METHOD

PROPERTY PUBLIC Size : UDINT
GET
Size := SIZEOF(activeData);
END_GET
END_PROPERTY

METHOD TryMakeReferenceTo : BOOL
VAR_INPUT
	Target : I_Datatype;
END_VAR
VAR
	targetAsEnum : I_EnumDatatype;
	pTargetData : POINTER TO ETcVnConnectedComponentsAlgorithm;
END_VAR
IF NOT Target.TryResolveAsEnumDatatype(targetAsEnum) THEN
	RETURN;
END_IF

IF targetAsEnum.Identifier <> Identifier THEN
	RETURN;
END_IF

pTargetData := Target.Address;
activeData REF= pTargetData^;
SetBaseDatatypeReference();
TryMakeReferenceTo := TRUE;
END_METHOD

PROPERTY PUBLIC Value : ETcVnConnectedComponentsAlgorithm
GET
Value := activeData;
END_GET
SET
activeData := Value;
END_SET
END_PROPERTY

END_FUNCTION_BLOCK

// Datatypes/Enums/_ETcVnContainerExportFormat
{attribute 'linkalways'} 
{attribute 'no_explicit_call' := 'This FB is a CLASS and must be accessed using methods or properties'}
{attribute 'enable_dynamic_creation'}
FUNCTION_BLOCK _ETcVnContainerExportFormat EXTENDS EnumDatatypeBase
VAR
	localData : ETcVnContainerExportFormat;
	activeData : REFERENCE TO ETcVnContainerExportFormat;
	enumBaseDatatype : _UINT(localData);
END_VAR

METHOD FB_init : BOOL
VAR_INPUT
	bInitRetains : BOOL; // if TRUE, the retain variables are initialized (warm start / cold start)
	bInCopyCode : BOOL;  // if TRUE, the instance afterwards gets moved into the copy code (online change)
	InitialValue : ETcVnContainerExportFormat;
END_VAR
localData := InitialValue;
AddBaseDatatype(enumBaseDatatype);
ClearReference();

AddLocalEnumeration('TCVN_CEF_XML', ETcVnContainerExportFormat.TCVN_CEF_XML);
AddLocalEnumeration('TCVN_CEF_XML_SERIALIZED', ETcVnContainerExportFormat.TCVN_CEF_XML_SERIALIZED);
AddLocalEnumeration('TCVN_CEF_CSV', ETcVnContainerExportFormat.TCVN_CEF_CSV);
AddLocalEnumeration('TCVN_CEF_BINARY', ETcVnContainerExportFormat.TCVN_CEF_BINARY);
END_METHOD

METHOD PRIVATE AddLocalEnumeration
VAR_INPUT
	Enumeration : T_MAXSTRING;
	Value : ETcVnContainerExportFormat;
END_VAR
AddEnumeration(Enumeration, Value);
END_METHOD

METHOD IsEnumeratorValueEqual : BOOL
VAR_INPUT
	Enumerator : I_KeyValueForwardEnumerator;
END_VAR
VAR
	storedValue : ETcVnContainerExportFormat;
END_VAR
IF NOT Enumerator.TryGet(storedValue) THEN
	RETURN;
END_IF

IsEnumeratorValueEqual := storedValue = activeData;
END_METHOD

METHOD PROTECTED SetBaseDatatypeReference
VAR_INPUT
END_VAR
enumBaseDatatype.MakeReferenceTo(activeData);
END_METHOD

PROPERTY PUBLIC Address : PVOID
GET
Address := ADR(activeData);
END_GET
END_PROPERTY

METHOD PUBLIC ClearReference
VAR_INPUT
END_VAR
activeData REF= localData;
SetBaseDatatypeReference();
END_METHOD

METHOD PUBLIC Clone : I_Datatype
VAR
    pClone : POINTER TO _ETcVnContainerExportFormat;
END_VAR
pClone := __NEW(_ETcVnContainerExportFormat(InitialValue := Value));
Clone := pClone^;
END_METHOD

PROPERTY PUBLIC Identifier : T_MAXSTRING
GET
Identifier := 'ETcVnContainerExportFormat';
END_GET
END_PROPERTY

METHOD PUBLIC MakeReferenceTo
VAR_INPUT
	ReferenceTarget : REFERENCE TO ETcVnContainerExportFormat;
END_VAR
activeData REF= ReferenceTarget;
SetBaseDatatypeReference();
END_METHOD

PROPERTY PUBLIC Size : UDINT
GET
Size := SIZEOF(activeData);
END_GET
END_PROPERTY

METHOD TryMakeReferenceTo : BOOL
VAR_INPUT
	Target : I_Datatype;
END_VAR
VAR
	targetAsEnum : I_EnumDatatype;
	pTargetData : POINTER TO ETcVnContainerExportFormat;
END_VAR
IF NOT Target.TryResolveAsEnumDatatype(targetAsEnum) THEN
	RETURN;
END_IF

IF targetAsEnum.Identifier <> Identifier THEN
	RETURN;
END_IF

pTargetData := Target.Address;
activeData REF= pTargetData^;
SetBaseDatatypeReference();
TryMakeReferenceTo := TRUE;
END_METHOD

PROPERTY PUBLIC Value : ETcVnContainerExportFormat
GET
Value := activeData;
END_GET
SET
activeData := Value;
END_SET
END_PROPERTY

END_FUNCTION_BLOCK

// Datatypes/Enums/_ETcVnContourApproximationMethod
{attribute 'linkalways'} 
{attribute 'no_explicit_call' := 'This FB is a CLASS and must be accessed using methods or properties'}
{attribute 'enable_dynamic_creation'}
FUNCTION_BLOCK _ETcVnContourApproximationMethod EXTENDS EnumDatatypeBase
VAR
	localData : ETcVnContourApproximationMethod;
	activeData : REFERENCE TO ETcVnContourApproximationMethod;
	enumBaseDatatype : _DINT(localData);
END_VAR

METHOD FB_init : BOOL
VAR_INPUT
	bInitRetains : BOOL; // if TRUE, the retain variables are initialized (warm start / cold start)
	bInCopyCode : BOOL;  // if TRUE, the instance afterwards gets moved into the copy code (online change)
	InitialValue : ETcVnContourApproximationMethod;
END_VAR
localData := InitialValue;
AddBaseDatatype(enumBaseDatatype);
ClearReference();

AddLocalEnumeration('TCVN_CAM_NONE', ETcVnContourApproximationMethod.TCVN_CAM_NONE);
AddLocalEnumeration('TCVN_CAM_SIMPLE', ETcVnContourApproximationMethod.TCVN_CAM_SIMPLE);
AddLocalEnumeration('TCVN_CAM_TC89_L1', ETcVnContourApproximationMethod.TCVN_CAM_TC89_L1);
AddLocalEnumeration('TCVN_CAM_TC89_KCOS', ETcVnContourApproximationMethod.TCVN_CAM_TC89_KCOS);
END_METHOD

METHOD PRIVATE AddLocalEnumeration
VAR_INPUT
	Enumeration : T_MAXSTRING;
	Value : ETcVnContourApproximationMethod;
END_VAR
AddEnumeration(Enumeration, Value);
END_METHOD

METHOD IsEnumeratorValueEqual : BOOL
VAR_INPUT
	Enumerator : I_KeyValueForwardEnumerator;
END_VAR
VAR
	storedValue : ETcVnContourApproximationMethod;
END_VAR
IF NOT Enumerator.TryGet(storedValue) THEN
	RETURN;
END_IF

IsEnumeratorValueEqual := storedValue = activeData;
END_METHOD

METHOD PROTECTED SetBaseDatatypeReference
VAR_INPUT
END_VAR
enumBaseDatatype.MakeReferenceTo(activeData);
END_METHOD

PROPERTY PUBLIC Address : PVOID
GET
Address := ADR(activeData);
END_GET
END_PROPERTY

METHOD PUBLIC ClearReference
VAR_INPUT
END_VAR
activeData REF= localData;
SetBaseDatatypeReference();
END_METHOD

METHOD PUBLIC Clone : I_Datatype
VAR
    pClone : POINTER TO _ETcVnContourApproximationMethod;
END_VAR
pClone := __NEW(_ETcVnContourApproximationMethod(InitialValue := Value));
Clone := pClone^;
END_METHOD

PROPERTY PUBLIC Identifier : T_MAXSTRING
GET
Identifier := 'ETcVnContourApproximationMethod';
END_GET
END_PROPERTY

METHOD PUBLIC MakeReferenceTo
VAR_INPUT
	ReferenceTarget : REFERENCE TO ETcVnContourApproximationMethod;
END_VAR
activeData REF= ReferenceTarget;
SetBaseDatatypeReference();
END_METHOD

PROPERTY PUBLIC Size : UDINT
GET
Size := SIZEOF(activeData);
END_GET
END_PROPERTY

METHOD TryMakeReferenceTo : BOOL
VAR_INPUT
	Target : I_Datatype;
END_VAR
VAR
	targetAsEnum : I_EnumDatatype;
	pTargetData : POINTER TO ETcVnContourApproximationMethod;
END_VAR
IF NOT Target.TryResolveAsEnumDatatype(targetAsEnum) THEN
	RETURN;
END_IF

IF targetAsEnum.Identifier <> Identifier THEN
	RETURN;
END_IF

pTargetData := Target.Address;
activeData REF= pTargetData^;
SetBaseDatatypeReference();
TryMakeReferenceTo := TRUE;
END_METHOD

PROPERTY PUBLIC Value : ETcVnContourApproximationMethod
GET
Value := activeData;
END_GET
SET
activeData := Value;
END_SET
END_PROPERTY

END_FUNCTION_BLOCK

// Datatypes/Enums/_ETcVnContourRetrievalMode
{attribute 'linkalways'} 
{attribute 'no_explicit_call' := 'This FB is a CLASS and must be accessed using methods or properties'}
{attribute 'enable_dynamic_creation'}
FUNCTION_BLOCK _ETcVnContourRetrievalMode EXTENDS EnumDatatypeBase
VAR
	localData : ETcVnContourRetrievalMode;
	activeData : REFERENCE TO ETcVnContourRetrievalMode;
	enumBaseDatatype : _DINT(localData);
END_VAR

METHOD FB_init : BOOL
VAR_INPUT
	bInitRetains : BOOL; // if TRUE, the retain variables are initialized (warm start / cold start)
	bInCopyCode : BOOL;  // if TRUE, the instance afterwards gets moved into the copy code (online change)
	InitialValue : ETcVnContourRetrievalMode;
END_VAR
localData := InitialValue;
AddBaseDatatype(enumBaseDatatype);
ClearReference();

AddLocalEnumeration('TCVN_CRM_EXTERNAL', ETcVnContourRetrievalMode.TCVN_CRM_EXTERNAL);
AddLocalEnumeration('TCVN_CRM_LIST', ETcVnContourRetrievalMode.TCVN_CRM_LIST);
AddLocalEnumeration('TCVN_CRM_CONNECTED_COMPONENTS', ETcVnContourRetrievalMode.TCVN_CRM_CONNECTED_COMPONENTS);
AddLocalEnumeration('TCVN_CRM_TREE', ETcVnContourRetrievalMode.TCVN_CRM_TREE);
AddLocalEnumeration('TCVN_CRM_FLOODFILL', ETcVnContourRetrievalMode.TCVN_CRM_FLOODFILL);
END_METHOD

METHOD PRIVATE AddLocalEnumeration
VAR_INPUT
	Enumeration : T_MAXSTRING;
	Value : ETcVnContourRetrievalMode;
END_VAR
AddEnumeration(Enumeration, Value);
END_METHOD

METHOD IsEnumeratorValueEqual : BOOL
VAR_INPUT
	Enumerator : I_KeyValueForwardEnumerator;
END_VAR
VAR
	storedValue : ETcVnContourRetrievalMode;
END_VAR
IF NOT Enumerator.TryGet(storedValue) THEN
	RETURN;
END_IF

IsEnumeratorValueEqual := storedValue = activeData;
END_METHOD

METHOD PROTECTED SetBaseDatatypeReference
VAR_INPUT
END_VAR
enumBaseDatatype.MakeReferenceTo(activeData);
END_METHOD

PROPERTY PUBLIC Address : PVOID
GET
Address := ADR(activeData);
END_GET
END_PROPERTY

METHOD PUBLIC ClearReference
VAR_INPUT
END_VAR
activeData REF= localData;
SetBaseDatatypeReference();
END_METHOD

METHOD PUBLIC Clone : I_Datatype
VAR
    pClone : POINTER TO _ETcVnContourRetrievalMode;
END_VAR
pClone := __NEW(_ETcVnContourRetrievalMode(InitialValue := Value));
Clone := pClone^;
END_METHOD

PROPERTY PUBLIC Identifier : T_MAXSTRING
GET
Identifier := 'ETcVnContourRetrievalMode';
END_GET
END_PROPERTY

METHOD PUBLIC MakeReferenceTo
VAR_INPUT
	ReferenceTarget : REFERENCE TO ETcVnContourRetrievalMode;
END_VAR
activeData REF= ReferenceTarget;
SetBaseDatatypeReference();
END_METHOD

PROPERTY PUBLIC Size : UDINT
GET
Size := SIZEOF(activeData);
END_GET
END_PROPERTY

METHOD TryMakeReferenceTo : BOOL
VAR_INPUT
	Target : I_Datatype;
END_VAR
VAR
	targetAsEnum : I_EnumDatatype;
	pTargetData : POINTER TO ETcVnContourRetrievalMode;
END_VAR
IF NOT Target.TryResolveAsEnumDatatype(targetAsEnum) THEN
	RETURN;
END_IF

IF targetAsEnum.Identifier <> Identifier THEN
	RETURN;
END_IF

pTargetData := Target.Address;
activeData REF= pTargetData^;
SetBaseDatatypeReference();
TryMakeReferenceTo := TRUE;
END_METHOD

PROPERTY PUBLIC Value : ETcVnContourRetrievalMode
GET
Value := activeData;
END_GET
SET
activeData := Value;
END_SET
END_PROPERTY

END_FUNCTION_BLOCK

// Datatypes/Enums/_ETcVnContoursMatchComparisonMethod
{attribute 'linkalways'} 
{attribute 'no_explicit_call' := 'This FB is a CLASS and must be accessed using methods or properties'}
{attribute 'enable_dynamic_creation'}
FUNCTION_BLOCK _ETcVnContoursMatchComparisonMethod EXTENDS EnumDatatypeBase
VAR
	localData : ETcVnContoursMatchComparisonMethod;
	activeData : REFERENCE TO ETcVnContoursMatchComparisonMethod;
	enumBaseDatatype : _DINT(localData);
END_VAR

METHOD FB_init : BOOL
VAR_INPUT
	bInitRetains : BOOL; // if TRUE, the retain variables are initialized (warm start / cold start)
	bInCopyCode : BOOL;  // if TRUE, the instance afterwards gets moved into the copy code (online change)
	InitialValue : ETcVnContoursMatchComparisonMethod;
END_VAR
localData := InitialValue;
AddBaseDatatype(enumBaseDatatype);
ClearReference();

AddLocalEnumeration('TCVN_CMCM_CONTOURS_MATCH_I1', ETcVnContoursMatchComparisonMethod.TCVN_CMCM_CONTOURS_MATCH_I1);
AddLocalEnumeration('TCVN_CMCM_CONTOURS_MATCH_I2', ETcVnContoursMatchComparisonMethod.TCVN_CMCM_CONTOURS_MATCH_I2);
AddLocalEnumeration('TCVN_CMCM_CONTOURS_MATCH_I3', ETcVnContoursMatchComparisonMethod.TCVN_CMCM_CONTOURS_MATCH_I3);
END_METHOD

METHOD PRIVATE AddLocalEnumeration
VAR_INPUT
	Enumeration : T_MAXSTRING;
	Value : ETcVnContoursMatchComparisonMethod;
END_VAR
AddEnumeration(Enumeration, Value);
END_METHOD

METHOD IsEnumeratorValueEqual : BOOL
VAR_INPUT
	Enumerator : I_KeyValueForwardEnumerator;
END_VAR
VAR
	storedValue : ETcVnContoursMatchComparisonMethod;
END_VAR
IF NOT Enumerator.TryGet(storedValue) THEN
	RETURN;
END_IF

IsEnumeratorValueEqual := storedValue = activeData;
END_METHOD

METHOD PROTECTED SetBaseDatatypeReference
VAR_INPUT
END_VAR
enumBaseDatatype.MakeReferenceTo(activeData);
END_METHOD

PROPERTY PUBLIC Address : PVOID
GET
Address := ADR(activeData);
END_GET
END_PROPERTY

METHOD PUBLIC ClearReference
VAR_INPUT
END_VAR
activeData REF= localData;
SetBaseDatatypeReference();
END_METHOD

METHOD PUBLIC Clone : I_Datatype
VAR
    pClone : POINTER TO _ETcVnContoursMatchComparisonMethod;
END_VAR
pClone := __NEW(_ETcVnContoursMatchComparisonMethod(InitialValue := Value));
Clone := pClone^;
END_METHOD

PROPERTY PUBLIC Identifier : T_MAXSTRING
GET
Identifier := 'ETcVnContoursMatchComparisonMethod';
END_GET
END_PROPERTY

METHOD PUBLIC MakeReferenceTo
VAR_INPUT
	ReferenceTarget : REFERENCE TO ETcVnContoursMatchComparisonMethod;
END_VAR
activeData REF= ReferenceTarget;
SetBaseDatatypeReference();
END_METHOD

PROPERTY PUBLIC Size : UDINT
GET
Size := SIZEOF(activeData);
END_GET
END_PROPERTY

METHOD TryMakeReferenceTo : BOOL
VAR_INPUT
	Target : I_Datatype;
END_VAR
VAR
	targetAsEnum : I_EnumDatatype;
	pTargetData : POINTER TO ETcVnContoursMatchComparisonMethod;
END_VAR
IF NOT Target.TryResolveAsEnumDatatype(targetAsEnum) THEN
	RETURN;
END_IF

IF targetAsEnum.Identifier <> Identifier THEN
	RETURN;
END_IF

pTargetData := Target.Address;
activeData REF= pTargetData^;
SetBaseDatatypeReference();
TryMakeReferenceTo := TRUE;
END_METHOD

PROPERTY PUBLIC Value : ETcVnContoursMatchComparisonMethod
GET
Value := activeData;
END_GET
SET
activeData := Value;
END_SET
END_PROPERTY

END_FUNCTION_BLOCK

// Datatypes/Enums/_ETcVnDiffusivityTypeKAZE
{attribute 'linkalways'} 
{attribute 'no_explicit_call' := 'This FB is a CLASS and must be accessed using methods or properties'}
{attribute 'enable_dynamic_creation'}
FUNCTION_BLOCK _ETcVnDiffusivityTypeKAZE EXTENDS EnumDatatypeBase
VAR
	localData : ETcVnDiffusivityTypeKAZE;
	activeData : REFERENCE TO ETcVnDiffusivityTypeKAZE;
	enumBaseDatatype : _DINT(localData);
END_VAR

METHOD FB_init : BOOL
VAR_INPUT
	bInitRetains : BOOL; // if TRUE, the retain variables are initialized (warm start / cold start)
	bInCopyCode : BOOL;  // if TRUE, the instance afterwards gets moved into the copy code (online change)
	InitialValue : ETcVnDiffusivityTypeKAZE;
END_VAR
localData := InitialValue;
AddBaseDatatype(enumBaseDatatype);
ClearReference();

AddLocalEnumeration('TCVN_DT1_KAZE_PM_G1', ETcVnDiffusivityTypeKAZE.TCVN_DT1_KAZE_PM_G1);
AddLocalEnumeration('TCVN_DT1_KAZE_PM_G2', ETcVnDiffusivityTypeKAZE.TCVN_DT1_KAZE_PM_G2);
AddLocalEnumeration('TCVN_DT1_KAZE_WEICKERT', ETcVnDiffusivityTypeKAZE.TCVN_DT1_KAZE_WEICKERT);
AddLocalEnumeration('TCVN_DT1_KAZE_CHARBONNIER', ETcVnDiffusivityTypeKAZE.TCVN_DT1_KAZE_CHARBONNIER);
END_METHOD

METHOD PRIVATE AddLocalEnumeration
VAR_INPUT
	Enumeration : T_MAXSTRING;
	Value : ETcVnDiffusivityTypeKAZE;
END_VAR
AddEnumeration(Enumeration, Value);
END_METHOD

METHOD IsEnumeratorValueEqual : BOOL
VAR_INPUT
	Enumerator : I_KeyValueForwardEnumerator;
END_VAR
VAR
	storedValue : ETcVnDiffusivityTypeKAZE;
END_VAR
IF NOT Enumerator.TryGet(storedValue) THEN
	RETURN;
END_IF

IsEnumeratorValueEqual := storedValue = activeData;
END_METHOD

METHOD PROTECTED SetBaseDatatypeReference
VAR_INPUT
END_VAR
enumBaseDatatype.MakeReferenceTo(activeData);
END_METHOD

PROPERTY PUBLIC Address : PVOID
GET
Address := ADR(activeData);
END_GET
END_PROPERTY

METHOD PUBLIC ClearReference
VAR_INPUT
END_VAR
activeData REF= localData;
SetBaseDatatypeReference();
END_METHOD

METHOD PUBLIC Clone : I_Datatype
VAR
    pClone : POINTER TO _ETcVnDiffusivityTypeKAZE;
END_VAR
pClone := __NEW(_ETcVnDiffusivityTypeKAZE(InitialValue := Value));
Clone := pClone^;
END_METHOD

PROPERTY PUBLIC Identifier : T_MAXSTRING
GET
Identifier := 'ETcVnDiffusivityTypeKAZE';
END_GET
END_PROPERTY

METHOD PUBLIC MakeReferenceTo
VAR_INPUT
	ReferenceTarget : REFERENCE TO ETcVnDiffusivityTypeKAZE;
END_VAR
activeData REF= ReferenceTarget;
SetBaseDatatypeReference();
END_METHOD

PROPERTY PUBLIC Size : UDINT
GET
Size := SIZEOF(activeData);
END_GET
END_PROPERTY

METHOD TryMakeReferenceTo : BOOL
VAR_INPUT
	Target : I_Datatype;
END_VAR
VAR
	targetAsEnum : I_EnumDatatype;
	pTargetData : POINTER TO ETcVnDiffusivityTypeKAZE;
END_VAR
IF NOT Target.TryResolveAsEnumDatatype(targetAsEnum) THEN
	RETURN;
END_IF

IF targetAsEnum.Identifier <> Identifier THEN
	RETURN;
END_IF

pTargetData := Target.Address;
activeData REF= pTargetData^;
SetBaseDatatypeReference();
TryMakeReferenceTo := TRUE;
END_METHOD

PROPERTY PUBLIC Value : ETcVnDiffusivityTypeKAZE
GET
Value := activeData;
END_GET
SET
activeData := Value;
END_SET
END_PROPERTY

END_FUNCTION_BLOCK

// Datatypes/Enums/_ETcVnDistanceTransformationLabel
{attribute 'linkalways'} 
{attribute 'no_explicit_call' := 'This FB is a CLASS and must be accessed using methods or properties'}
{attribute 'enable_dynamic_creation'}
FUNCTION_BLOCK _ETcVnDistanceTransformationLabel EXTENDS EnumDatatypeBase
VAR
	localData : ETcVnDistanceTransformationLabel;
	activeData : REFERENCE TO ETcVnDistanceTransformationLabel;
	enumBaseDatatype : _DINT(localData);
END_VAR

